C03659=1114.232,220.895,-68.578,-178.796,9.608,149.566
C03660=1114.228,221.144,-68.604,-178.794,9.611,149.566
C03661=1114.223,221.393,-68.631,-178.792,9.614,149.567
C03662=1114.219,221.641,-68.657,-178.789,9.617,149.567
C03663=1114.214,221.890,-68.684,-178.787,9.620,149.567
C03664=1114.210,222.138,-68.710,-178.784,9.623,149.567
C03665=1114.206,222.387,-68.737,-178.782,9.626,149.567
C03666=1114.202,222.635,-68.764,-178.779,9.629,149.567
C03667=1114.197,222.884,-68.790,-178.777,9.632,149.567
C03668=1114.193,223.132,-68.816,-178.774,9.635,149.567
C03669=1114.188,223.381,-68.843,-178.772,9.638,149.567
C03670=1114.184,223.629,-68.869,-178.769,9.642,149.567
C03671=1114.179,223.878,-68.896,-178.767,9.645,149.567
C03672=1114.175,224.126,-68.923,-178.764,9.648,149.567
C03673=1114.171,224.375,-68.950,-178.762,9.651,149.567
C03674=1114.166,224.623,-68.977,-178.759,9.654,149.567
C03675=1114.162,224.872,-69.003,-178.755,9.657,149.567
C03676=1114.157,225.120,-69.030,-178.753,9.661,149.567
C03677=1114.153,225.369,-69.057,-178.750,9.664,149.567
C03678=1114.150,225.582,-69.080,-178.749,9.666,149.567
C03679=1114.146,225.795,-69.102,-178.746,9.669,149.568
C03680=1114.142,226.008,-69.126,-178.744,9.671,149.568
C03681=1114.138,226.222,-69.149,-178.741,9.674,149.567
C03682=1114.135,226.435,-69.172,-178.739,9.677,149.568
C03683=1114.131,226.648,-69.194,-178.737,9.680,149.568
C03684=1114.127,226.861,-69.218,-178.735,9.682,149.568
C03685=1114.123,227.074,-69.241,-178.732,9.685,149.568
C03686=1114.119,227.323,-69.268,-178.729,9.688,149.568
C03687=1114.114,227.572,-69.294,-178.727,9.691,149.568
C03688=1114.110,227.820,-69.321,-178.724,9.694,149.568
C03689=1114.105,228.069,-69.348,-178.721,9.697,149.568
C03690=1114.101,228.317,-69.375,-178.718,9.700,149.567
C03691=1114.097,228.565,-69.403,-178.715,9.703,149.568
C03692=1114.093,228.814,-69.430,-178.712,9.706,149.567
C03693=1114.088,229.062,-69.457,-178.710,9.709,149.568
C03694=1114.084,229.311,-69.484,-178.707,9.712,149.567
C03695=1114.080,229.559,-69.511,-178.704,9.715,149.567
C03696=1114.075,229.808,-69.538,-178.701,9.719,149.567
C03697=1114.070,230.056,-69.565,-178.698,9.721,149.567
C03698=1114.066,230.305,-69.592,-178.695,9.724,149.567
C03699=1114.062,230.553,-69.619,-178.692,9.727,149.567
C03700=1114.058,230.802,-69.646,-178.689,9.730,149.567
C03701=1114.053,231.050,-69.673,-178.686,9.733,149.567
C03702=1114.049,231.298,-69.701,-178.684,9.736,149.567
C03703=1114.045,231.547,-69.728,-178.680,9.739,149.567
C03704=1114.040,231.796,-69.755,-178.677,9.742,149.567
C03705=1114.036,232.044,-69.781,-178.674,9.745,149.567
C03706=1114.032,232.292,-69.809,-178.672,9.748,149.566
C03707=1114.028,232.541,-69.837,-178.669,9.751,149.567
C03708=1114.023,232.790,-69.864,-178.666,9.754,149.566
C03709=1114.018,233.038,-69.891,-178.663,9.756,149.566
C03710=1114.014,233.286,-69.919,-178.661,9.758,149.566
C03711=1114.010,233.535,-69.946,-178.658,9.761,149.566
C03712=1114.005,233.784,-69.973,-178.655,9.764,149.566
C03713=1114.001,234.032,-70.001,-178.652,9.767,149.566
C03714=1113.997,234.281,-70.028,-178.649,9.770,149.566
C03715=1113.992,234.529,-70.055,-178.646,9.772,149.566
C03716=1113.989,234.777,-70.083,-178.644,9.775,149.566
C03717=1113.984,235.025,-70.110,-178.641,9.778,149.565
C03718=1113.980,235.274,-70.138,-178.639,9.780,149.566
C03719=1113.975,235.522,-70.165,-178.636,9.783,149.565
C03720=1113.971,235.771,-70.192,-178.633,9.786,149.565
C03721=1113.967,236.020,-70.220,-178.630,9.788,149.565
C03722=1113.962,236.268,-70.247,-178.627,9.791,149.565
C03723=1113.958,236.516,-70.275,-178.625,9.794,149.565
C03724=1113.954,236.765,-70.302,-178.622,9.796,149.565
C03725=1113.950,237.013,-70.330,-178.619,9.799,149.565
C03726=1113.944,237.262,-70.358,-178.617,9.801,149.565
C03727=1113.941,237.510,-70.386,-178.614,9.804,149.565
C03728=1113.936,237.759,-70.413,-178.611,9.807,149.565
C03729=1113.932,238.007,-70.441,-178.608,9.810,149.565
C03730=1113.927,238.256,-70.468,-178.606,9.812,149.564
C03731=1113.923,238.504,-70.496,-178.603,9.814,149.564
C03732=1113.919,238.752,-70.524,-178.601,9.816,149.564
C03733=1113.915,239.001,-70.551,-178.598,9.819,149.564
C03734=1113.911,239.214,-70.575,-178.596,9.821,149.564
C03735=1113.907,239.427,-70.598,-178.594,9.823,149.564
C03736=1113.903,239.640,-70.623,-178.592,9.826,149.564
C03737=1113.899,239.853,-70.646,-178.589,9.828,149.564
C03738=1113.896,240.066,-70.670,-178.587,9.831,149.564
C03739=1113.892,240.279,-70.694,-178.585,9.833,149.564
C03740=1113.889,240.492,-70.718,-178.583,9.835,149.564
C03741=1113.885,240.705,-70.742,-178.580,9.837,149.564
C03742=1113.880,240.954,-70.769,-178.578,9.839,149.564
C03743=1113.876,241.202,-70.797,-178.576,9.842,149.564
C03744=1113.872,241.450,-70.825,-178.573,9.844,149.564
C03745=1113.868,241.699,-70.853,-178.571,9.847,149.564
C03746=1113.863,241.947,-70.880,-178.568,9.849,149.563
C03747=1113.859,242.195,-70.908,-178.566,9.852,149.564
C03748=1113.855,242.444,-70.937,-178.564,9.854,149.563
C03749=1113.850,242.692,-70.965,-178.561,9.857,149.563
C03750=1113.846,242.941,-70.992,-178.559,9.859,149.563
C03751=1113.842,243.189,-71.020,-178.556,9.863,149.563
C03752=1113.837,243.438,-71.049,-178.554,9.864,149.563
C03753=1113.833,243.686,-71.076,-178.551,9.868,149.563
C03754=1113.829,243.934,-71.104,-178.549,9.870,149.563
C03755=1113.825,244.183,-71.131,-178.547,9.873,149.563
C03756=1113.820,244.432,-71.160,-178.545,9.875,149.563
C03757=1113.816,244.679,-71.188,-178.542,9.878,149.563
C03758=1113.812,244.928,-71.216,-178.540,9.880,149.563
C03759=1113.808,245.176,-71.244,-178.538,9.882,149.563
C03760=1113.803,245.425,-71.273,-178.535,9.886,149.563
C03761=1113.799,245.673,-71.300,-178.533,9.888,149.564
C03762=1113.795,245.921,-71.329,-178.531,9.891,149.563
C03763=1113.790,246.169,-71.357,-178.529,9.893,149.563
C03764=1113.786,246.418,-71.385,-178.526,9.896,149.564
C03765=1113.782,246.666,-71.413,-178.524,9.898,149.564
C03766=1113.777,246.915,-71.441,-178.522,9.901,149.564
C03767=1113.773,247.163,-71.469,-178.520,9.904,149.564
C03768=1113.769,247.412,-71.497,-178.518,9.906,149.564
C03769=1113.764,247.660,-71.525,-178.514,9.910,149.564
C03770=1113.760,247.909,-71.553,-178.511,9.913,149.564
C03771=1113.755,248.156,-71.582,-178.507,9.918,149.564
C03772=1113.752,248.405,-71.611,-178.503,9.921,149.563
C03773=1113.748,248.653,-71.639,-178.499,9.924,149.563
C03774=1113.743,248.902,-71.667,-178.495,9.927,149.563
C03775=1113.739,249.150,-71.695,-178.491,9.931,149.563
C03776=1113.734,249.398,-71.724,-178.487,9.934,149.562
C03777=1113.730,249.647,-71.752,-178.484,9.937,149.562
C03778=1113.726,249.896,-71.780,-178.481,9.940,149.562
C03779=1113.721,250.144,-71.808,-178.477,9.942,149.562
C03780=1113.717,250.392,-71.838,-178.474,9.946,149.562
C03781=1113.713,250.640,-71.865,-178.470,9.948,149.561
C03782=1113.708,250.889,-71.894,-178.467,9.951,149.561
C03783=1113.705,251.137,-71.922,-178.464,9.954,149.561
C03784=1113.700,251.385,-71.951,-178.461,9.956,149.561
C03785=1113.696,251.633,-71.980,-178.458,9.959,149.561
C03786=1113.692,251.882,-72.008,-178.455,9.961,149.560
C03787=1113.687,252.130,-72.036,-178.452,9.964,149.560
C03788=1113.683,252.378,-72.066,-178.449,9.967,149.560
C03789=1113.679,252.627,-72.094,-178.446,9.969,149.560
C03790=1113.675,252.840,-72.119,-178.444,9.971,149.560
C03791=1113.672,253.052,-72.143,-178.442,9.973,149.560
C03792=1113.668,253.266,-72.168,-178.440,9.975,149.560
C03793=1113.664,253.479,-72.192,-178.437,9.977,149.560
C03794=1113.660,253.691,-72.216,-178.435,9.979,149.559
C03795=1113.657,253.905,-72.241,-178.433,9.981,149.559
C03796=1113.653,254.117,-72.266,-178.431,9.982,149.559
C03797=1113.649,254.330,-72.290,-178.429,9.984,149.559
C03798=1113.645,254.578,-72.319,-178.427,9.987,149.559
C03799=1113.641,254.827,-72.348,-178.425,9.989,149.559
C03800=1113.637,255.076,-72.377,-178.423,9.991,149.559
C03801=1113.633,255.323,-72.405,-178.421,9.993,149.559
C03802=1113.628,255.572,-72.434,-178.420,9.995,149.559
C03803=1113.624,255.821,-72.463,-178.418,9.997,149.559
C03804=1113.620,256.068,-72.491,-178.416,10.000,149.559
C03805=1113.615,256.317,-72.520,-178.413,10.002,149.559
C03806=1113.611,256.565,-72.549,-178.410,10.005,149.559
C03807=1113.607,256.814,-72.578,-178.408,10.007,149.559
C03808=1113.602,257.061,-72.607,-178.405,10.010,149.559
C03809=1113.598,257.310,-72.635,-178.402,10.013,149.559
C03810=1113.594,257.558,-72.665,-178.399,10.016,149.559
C03811=1113.590,257.806,-72.694,-178.396,10.018,149.559
C03812=1113.585,258.054,-72.722,-178.394,10.022,149.559
C03813=1113.581,258.303,-72.752,-178.391,10.024,149.559
C03814=1113.577,258.551,-72.780,-178.388,10.027,149.559
C03815=1113.573,258.800,-72.809,-178.385,10.030,149.559
C03816=1113.569,259.048,-72.839,-178.382,10.033,149.558
C03817=1113.564,259.296,-72.867,-178.379,10.035,149.558
C03818=1113.560,259.544,-72.896,-178.376,10.038,149.558
C03819=1113.556,259.793,-72.925,-178.374,10.041,149.558
C03820=1113.552,260.041,-72.954,-178.371,10.044,149.558
C03821=1113.548,260.289,-72.983,-178.368,10.047,149.558
C03822=1113.543,260.537,-73.013,-178.365,10.049,149.558
C03823=1113.538,260.786,-73.041,-178.362,10.052,149.558
C03824=1113.535,261.034,-73.070,-178.359,10.055,149.558
C03825=1113.531,261.282,-73.100,-178.356,10.058,149.558
C03826=1113.526,261.530,-73.129,-178.353,10.060,149.558
C03827=1113.522,261.779,-73.158,-178.350,10.063,149.558
C03828=1113.518,262.027,-73.187,-178.347,10.066,149.557
C03829=1113.513,262.275,-73.216,-178.344,10.068,149.557
C03830=1113.509,262.523,-73.246,-178.341,10.071,149.557
C03831=1113.505,262.772,-73.275,-178.338,10.074,149.557
C03832=1113.501,263.020,-73.303,-178.335,10.077,149.557
C03833=1113.497,263.268,-73.333,-178.332,10.080,149.557
C03834=1113.493,263.517,-73.362,-178.328,10.083,149.556
C03835=1113.488,263.765,-73.392,-178.325,10.085,149.556
C03836=1113.484,264.013,-73.421,-178.322,10.088,149.556
C03837=1113.479,264.261,-73.450,-178.319,10.091,149.556
C03838=1113.475,264.509,-73.480,-178.316,10.093,149.556
C03839=1113.471,264.757,-73.509,-178.313,10.096,149.556
C03840=1113.467,265.006,-73.539,-178.311,10.098,149.556
C03841=1113.463,265.254,-73.568,-178.308,10.101,149.555
C03842=1113.458,265.502,-73.598,-178.305,10.104,149.555
C03843=1113.454,265.750,-73.627,-178.303,10.106,149.555
C03844=1113.450,265.999,-73.656,-178.300,10.108,149.555
C03845=1113.446,266.247,-73.686,-178.297,10.111,149.555
C03846=1113.442,266.460,-73.711,-178.294,10.113,149.555
C03847=1113.438,266.672,-73.737,-178.292,10.115,149.555
C03848=1113.434,266.885,-73.761,-178.290,10.117,149.555
C03849=1113.431,267.098,-73.787,-178.288,10.119,149.555
C03850=1113.427,267.311,-73.813,-178.285,10.122,149.554
C03851=1113.424,267.523,-73.838,-178.282,10.124,149.554
C03852=1113.420,267.737,-73.863,-178.280,10.126,149.554
C03853=1113.416,267.949,-73.889,-178.278,10.128,149.554
C03854=1113.412,268.197,-73.918,-178.275,10.131,149.554
C03855=1113.408,268.445,-73.948,-178.272,10.134,149.554
C03856=1113.404,268.694,-73.977,-178.270,10.136,149.554
C03857=1113.399,268.942,-74.007,-178.267,10.138,149.554
C03858=1113.395,269.190,-74.036,-178.264,10.141,149.554
C03859=1113.391,269.438,-74.066,-178.261,10.144,149.554
C03860=1113.387,269.686,-74.096,-178.259,10.146,149.553
C03861=1113.382,269.935,-74.126,-178.256,10.149,149.553
C03862=1113.378,270.183,-74.155,-178.253,10.151,149.553
C03863=1113.374,270.431,-74.185,-178.250,10.154,149.553
C03864=1113.370,270.679,-74.215,-178.247,10.156,149.553
C03865=1113.366,270.927,-74.244,-178.244,10.158,149.553
C03866=1113.362,271.176,-74.275,-178.241,10.161,149.553
C03867=1113.358,271.424,-74.305,-178.238,10.164,149.553
C03868=1113.354,271.672,-74.334,-178.235,10.167,149.552
C03869=1113.349,271.921,-74.364,-178.233,10.170,149.552
C03870=1113.345,272.168,-74.394,-178.230,10.172,149.552
C03871=1113.341,272.417,-74.424,-178.227,10.174,149.552
C03872=1113.336,272.665,-74.453,-178.224,10.177,149.552
C03873=1113.333,272.913,-74.484,-178.221,10.180,149.552
C03874=1113.328,273.161,-74.513,-178.219,10.183,149.552
C03875=1113.323,273.410,-74.543,-178.216,10.185,149.552
C03876=1113.320,273.657,-74.573,-178.213,10.188,149.552
C03877=1113.315,273.906,-74.603,-178.210,10.191,149.552
C03878=1113.312,274.154,-74.633,-178.206,10.193,149.551
C03879=1113.307,274.402,-74.663,-178.204,10.195,149.551
C03880=1113.303,274.650,-74.693,-178.201,10.198,149.551
C03881=1113.299,274.898,-74.723,-178.198,10.201,149.551
C03882=1113.294,275.146,-74.754,-178.195,10.204,149.551
C03883=1113.290,275.395,-74.783,-178.192,10.206,149.551
C03884=1113.286,275.642,-74.813,-178.189,10.209,149.551
C03885=1113.282,275.892,-74.844,-178.186,10.211,149.550
C03886=1113.278,276.139,-74.874,-178.183,10.214,149.550
C03887=1113.274,276.387,-74.903,-178.180,10.217,149.550
C03888=1113.269,276.635,-74.934,-178.177,10.220,149.550
C03889=1113.266,276.883,-74.964,-178.174,10.223,149.550
C03890=1113.261,277.131,-74.994,-178.171,10.225,149.550
C03891=1113.257,277.380,-75.025,-178.168,10.228,149.550
C03892=1113.253,277.628,-75.055,-178.165,10.230,149.550
C03893=1113.249,277.876,-75.085,-178.163,10.232,149.549
C03894=1113.245,278.124,-75.115,-178.159,10.235,149.549
C03895=1113.240,278.372,-75.146,-178.156,10.238,149.549
C03896=1113.237,278.621,-75.176,-178.154,10.240,149.549
C03897=1113.233,278.868,-75.206,-178.150,10.243,149.549
C03898=1113.228,279.116,-75.237,-178.147,10.246,149.549
C03899=1113.224,279.365,-75.266,-178.144,10.248,149.548
C03900=1113.220,279.613,-75.297,-178.141,10.251,149.548
C03901=1113.216,279.861,-75.327,-178.138,10.253,149.548
C03902=1113.212,280.074,-75.354,-178.135,10.256,149.548
C03903=1113.208,280.286,-75.380,-178.133,10.258,149.548
C03904=1113.205,280.499,-75.405,-178.130,10.260,149.548
C03905=1113.201,280.712,-75.432,-178.127,10.263,149.547
C03906=1113.198,280.924,-75.459,-178.125,10.265,149.547
C03907=1113.194,281.136,-75.484,-178.122,10.267,149.547
C03908=1113.190,281.349,-75.511,-178.120,10.269,149.547
C03909=1113.187,281.562,-75.536,-178.116,10.272,149.547
C03910=1113.183,281.810,-75.567,-178.114,10.274,149.547
C03911=1113.179,282.059,-75.598,-178.111,10.276,149.546
C03912=1113.174,282.306,-75.628,-178.108,10.279,149.546
C03913=1113.170,282.554,-75.659,-178.105,10.282,149.546
C03914=1113.166,282.802,-75.689,-178.101,10.284,149.546
C03915=1113.162,283.051,-75.721,-178.098,10.287,149.546
C03916=1113.158,283.299,-75.750,-178.095,10.289,149.546
C03917=1113.153,283.547,-75.781,-178.092,10.292,149.546
C03918=1113.150,283.795,-75.811,-178.090,10.294,149.545
C03919=1113.145,284.043,-75.842,-178.087,10.296,149.545
C03920=1113.140,284.291,-75.873,-178.084,10.299,149.545
C03921=1113.137,284.540,-75.903,-178.080,10.302,149.545
C03922=1113.133,284.787,-75.935,-178.077,10.304,149.545
C03923=1113.128,285.035,-75.966,-178.074,10.307,149.544
C03924=1113.125,285.283,-75.996,-178.071,10.310,149.544
C03925=1113.120,285.531,-76.027,-178.068,10.312,149.544
C03926=1113.116,285.779,-76.058,-178.065,10.315,149.544
C03927=1113.112,286.028,-76.089,-178.062,10.317,149.544
C03928=1113.108,286.275,-76.119,-178.059,10.319,149.544
C03929=1113.104,286.524,-76.150,-178.056,10.322,149.543
C03930=1113.099,286.772,-76.181,-178.053,10.324,149.543
C03931=1113.096,287.019,-76.212,-178.050,10.327,149.543
C03932=1113.092,287.268,-76.243,-178.047,10.330,149.543
C03933=1113.087,287.516,-76.274,-178.044,10.332,149.543
C03934=1113.083,287.764,-76.305,-178.041,10.335,149.543
C03935=1113.078,288.012,-76.336,-178.038,10.337,149.542
C03936=1113.075,288.259,-76.366,-178.035,10.340,149.542
C03937=1113.071,288.508,-76.398,-178.032,10.342,149.542
C03938=1113.066,288.756,-76.428,-178.029,10.345,149.542
C03939=1113.062,289.005,-76.459,-178.026,10.347,149.542
C03940=1113.058,289.252,-76.491,-178.023,10.350,149.542
C03941=1113.055,289.500,-76.521,-178.020,10.353,149.541
C03942=1113.050,289.748,-76.552,-178.016,10.355,149.541
C03943=1113.046,289.996,-76.584,-178.013,10.358,149.541
C03944=1113.042,290.244,-76.615,-178.011,10.359,149.541
C03945=1113.037,290.492,-76.646,-178.008,10.362,149.541
C03946=1113.033,290.740,-76.677,-178.004,10.365,149.540
C03947=1113.029,290.988,-76.708,-178.001,10.367,149.540
C03948=1113.026,291.236,-76.739,-177.998,10.370,149.540
C03949=1113.021,291.484,-76.770,-177.995,10.373,149.540
C03950=1113.017,291.733,-76.801,-177.992,10.375,149.540
C03951=1113.013,291.980,-76.833,-177.989,10.378,149.540
C03952=1113.009,292.229,-76.864,-177.986,10.381,149.540
C03953=1113.005,292.476,-76.895,-177.983,10.382,149.539
C03954=1113.001,292.725,-76.927,-177.980,10.385,149.539
C03955=1112.997,292.973,-76.958,-177.977,10.387,149.539
C03956=1112.992,293.221,-76.989,-177.974,10.390,149.539
C03957=1112.989,293.469,-77.021,-177.971,10.393,149.539
C03958=1112.985,293.681,-77.048,-177.968,10.395,149.538
C03959=1112.982,293.894,-77.074,-177.965,10.397,149.538
C03960=1112.978,294.106,-77.101,-177.963,10.399,149.538
C03961=1112.974,294.319,-77.129,-177.960,10.401,149.538
C03962=1112.971,294.531,-77.155,-177.958,10.404,149.538
C03963=1112.968,294.743,-77.182,-177.955,10.406,149.538
C03964=1112.964,294.956,-77.210,-177.953,10.408,149.538
C03965=1112.961,295.169,-77.235,-177.950,10.410,149.537
C03966=1112.956,295.416,-77.267,-177.947,10.413,149.537
C03967=1112.953,295.664,-77.299,-177.944,10.415,149.537
C03968=1112.947,295.912,-77.330,-177.941,10.417,149.537
C03969=1112.944,296.160,-77.362,-177.938,10.420,149.537
C03970=1112.940,296.408,-77.394,-177.935,10.423,149.537
C03971=1112.935,296.656,-77.425,-177.932,10.425,149.536
C03972=1112.932,296.904,-77.456,-177.928,10.428,149.536
C03973=1112.927,297.152,-77.488,-177.926,10.431,149.536
C03974=1112.924,297.400,-77.520,-177.922,10.433,149.536
C03975=1112.920,297.648,-77.551,-177.919,10.436,149.536
C03976=1112.915,297.896,-77.582,-177.917,10.437,149.535
C03977=1112.911,298.144,-77.615,-177.914,10.440,149.535
C03978=1112.907,298.392,-77.647,-177.910,10.443,149.535
C03979=1112.903,298.640,-77.678,-177.907,10.445,149.535
C03980=1112.899,298.888,-77.709,-177.904,10.448,149.535
C03981=1112.895,299.136,-77.741,-177.901,10.451,149.535
C03982=1112.891,299.384,-77.773,-177.898,10.453,149.534
C03983=1112.886,299.632,-77.805,-177.895,10.456,149.534
C03984=1112.883,299.880,-77.837,-177.892,10.458,149.534
C03985=1112.878,300.127,-77.868,-177.889,10.461,149.534
C03986=1112.875,300.375,-77.900,-177.886,10.463,149.534
C03987=1112.871,300.623,-77.932,-177.883,10.465,149.534
C03988=1112.866,300.871,-77.964,-177.880,10.468,149.533
C03989=1112.862,301.119,-77.996,-177.877,10.471,149.533
C03990=1112.858,301.367,-78.028,-177.873,10.473,149.533
C03991=1112.853,301.615,-78.060,-177.870,10.476,149.533
C03992=1112.850,301.863,-78.092,-177.867,10.478,149.533
C03993=1112.846,302.111,-78.124,-177.864,10.481,149.533
C03994=1112.842,302.358,-78.155,-177.861,10.483,149.532
C03995=1112.837,302.607,-78.188,-177.859,10.485,149.532
C03996=1112.833,302.855,-78.219,-177.855,10.488,149.532
C03997=1112.830,303.103,-78.251,-177.852,10.491,149.532
C03998=1112.825,303.350,-78.283,-177.849,10.493,149.532
C03999=1112.821,303.598,-78.315,-177.846,10.496,149.532
C04000=1112.817,303.847,-78.348,-177.843,10.498,149.531
C04001=1112.813,304.095,-78.379,-177.840,10.501,149.531
C04002=1112.809,304.342,-78.411,-177.836,10.503,149.531
C04003=1112.804,304.590,-78.443,-177.833,10.506,149.531
C04004=1112.801,304.838,-78.476,-177.830,10.509,149.531
C04005=1112.797,305.086,-78.508,-177.827,10.510,149.530
C04006=1112.792,305.333,-78.540,-177.825,10.513,149.530
C04007=1112.788,305.582,-78.572,-177.821,10.516,149.530
C04008=1112.784,305.830,-78.604,-177.818,10.518,149.530
C04009=1112.780,306.077,-78.637,-177.815,10.521,149.530
C04010=1112.776,306.326,-78.669,-177.812,10.523,149.530
C04011=1112.772,306.573,-78.701,-177.809,10.526,149.529
C04012=1112.768,306.821,-78.732,-177.806,10.529,149.529
C04013=1112.764,307.069,-78.766,-177.802,10.531,149.529
C04014=1112.760,307.281,-78.793,-177.800,10.533,149.529
C04015=1112.757,307.493,-78.821,-177.798,10.535,149.529
C04016=1112.754,307.706,-78.848,-177.794,10.538,149.528
C04017=1112.750,307.918,-78.876,-177.792,10.540,149.528
C04018=1112.747,308.131,-78.903,-177.790,10.542,149.528
C04019=1112.742,308.343,-78.932,-177.787,10.544,149.528
C04020=1112.739,308.556,-78.959,-177.784,10.546,149.528
C04021=1112.736,308.768,-78.987,-177.782,10.548,149.528
C04022=1112.732,309.016,-79.019,-177.779,10.550,149.528
C04023=1112.728,309.264,-79.052,-177.776,10.553,149.527
C04024=1112.724,309.511,-79.084,-177.772,10.556,149.527
C04025=1112.719,309.759,-79.116,-177.769,10.558,149.527
C04026=1112.716,310.007,-79.149,-177.766,10.561,149.527
C04027=1112.712,310.255,-79.181,-177.763,10.563,149.527
C04028=1112.707,310.503,-79.214,-177.760,10.566,149.527
C04029=1112.704,310.751,-79.246,-177.757,10.568,149.526
C04030=1112.700,310.999,-79.279,-177.754,10.570,149.526
C04031=1112.696,311.247,-79.311,-177.751,10.573,149.526
C04032=1112.692,311.494,-79.345,-177.748,10.576,149.526
C04033=1112.687,311.743,-79.377,-177.745,10.578,149.526
C04034=1112.684,311.990,-79.410,-177.741,10.581,149.525
C04035=1112.679,312.237,-79.442,-177.738,10.583,149.525
C04036=1112.675,312.485,-79.475,-177.735,10.586,149.525
C04037=1112.671,312.733,-79.507,-177.732,10.589,149.525
C04038=1112.667,312.981,-79.540,-177.729,10.591,149.525
C04039=1112.663,313.229,-79.573,-177.726,10.594,149.525
C04040=1112.659,313.476,-79.605,-177.723,10.595,149.524
C04041=1112.655,313.725,-79.638,-177.720,10.598,149.524
C04042=1112.651,313.972,-79.671,-177.717,10.601,149.524
C04043=1112.647,314.220,-79.704,-177.714,10.603,149.524
C04044=1112.643,314.468,-79.737,-177.711,10.606,149.524
C04045=1112.639,314.716,-79.769,-177.707,10.608,149.523
C04046=1112.635,314.963,-79.802,-177.704,10.611,149.523
C04047=1112.631,315.211,-79.835,-177.701,10.613,149.523
C04048=1112.627,315.459,-79.868,-177.698,10.616,149.523
C04049=1112.623,315.707,-79.901,-177.695,10.619,149.523
C04050=1112.619,315.955,-79.933,-177.692,10.620,149.523
C04051=1112.615,316.202,-79.966,-177.689,10.623,149.522
C04052=1112.611,316.450,-79.999,-177.686,10.626,149.522
C04053=1112.607,316.698,-80.033,-177.683,10.628,149.522
C04054=1112.603,316.946,-80.066,-177.680,10.631,149.522
C04055=1112.599,317.194,-80.098,-177.676,10.633,149.522
C04056=1112.595,317.441,-80.131,-177.673,10.636,149.522
C04057=1112.591,317.690,-80.164,-177.670,10.638,149.521
C04058=1112.587,317.937,-80.197,-177.667,10.641,149.521
C04059=1112.583,318.185,-80.231,-177.664,10.644,149.521
C04060=1112.579,318.433,-80.264,-177.660,10.646,149.521
C04061=1112.575,318.680,-80.296,-177.658,10.648,149.521
C04062=1112.571,318.928,-80.329,-177.655,10.651,149.520
C04063=1112.567,319.176,-80.363,-177.652,10.653,149.520
C04064=1112.563,319.424,-80.396,-177.649,10.656,149.520
C04065=1112.559,319.671,-80.429,-177.645,10.658,149.520
C04066=1112.555,319.919,-80.462,-177.642,10.661,149.520
C04067=1112.551,320.167,-80.496,-177.639,10.663,149.520
C04068=1112.547,320.415,-80.529,-177.636,10.666,149.519
C04069=1112.544,320.663,-80.561,-177.633,10.669,149.519
C04070=1112.540,320.875,-80.590,-177.630,10.670,149.519
C04071=1112.537,321.087,-80.618,-177.628,10.672,149.519
C04072=1112.533,321.299,-80.647,-177.624,10.675,149.519
C04073=1112.530,321.511,-80.676,-177.622,10.677,149.518
C04074=1112.526,321.724,-80.704,-177.620,10.679,149.518
C04075=1112.523,321.936,-80.732,-177.617,10.681,149.518
C04076=1112.519,322.148,-80.761,-177.614,10.683,149.518
C04077=1112.516,322.360,-80.790,-177.612,10.685,149.518
C04078=1112.513,322.608,-80.823,-177.609,10.688,149.518
C04079=1112.508,322.856,-80.856,-177.605,10.690,149.517
C04080=1112.504,323.103,-80.889,-177.602,10.693,149.517
C04081=1112.500,323.351,-80.923,-177.599,10.695,149.517
C04082=1112.496,323.598,-80.956,-177.596,10.698,149.517
C04083=1112.493,323.847,-80.990,-177.593,10.701,149.517
C04084=1112.489,324.094,-81.023,-177.590,10.703,149.517
C04085=1112.485,324.342,-81.056,-177.586,10.705,149.516
C04086=1112.480,324.590,-81.091,-177.583,10.708,149.516
C04087=1112.476,324.837,-81.124,-177.581,10.710,149.516
C04088=1112.472,325.086,-81.157,-177.577,10.712,149.516
C04089=1112.468,325.333,-81.191,-177.574,10.715,149.516
C04090=1112.464,325.581,-81.224,-177.571,10.718,149.515
C04091=1112.460,325.828,-81.258,-177.568,10.720,149.515
C04092=1112.457,326.076,-81.292,-177.565,10.723,149.515
C04093=1112.453,326.324,-81.325,-177.561,10.725,149.515
C04094=1112.449,326.571,-81.359,-177.558,10.728,149.515
C04095=1112.444,326.819,-81.393,-177.555,10.730,149.515
C04096=1112.441,327.067,-81.426,-177.552,10.733,149.514
C04097=1112.437,327.315,-81.460,-177.549,10.735,149.514
C04098=1112.433,327.562,-81.493,-177.546,10.737,149.514
C04099=1112.429,327.809,-81.527,-177.543,10.740,149.514
C04100=1112.425,328.058,-81.561,-177.540,10.742,149.514
C04101=1112.421,328.305,-81.595,-177.537,10.745,149.513
C04102=1112.417,328.553,-81.628,-177.533,10.747,149.513
C04103=1112.413,328.800,-81.662,-177.530,10.750,149.513
C04104=1112.409,329.048,-81.696,-177.527,10.753,149.513
C04105=1112.405,329.296,-81.730,-177.524,10.755,149.513
C04106=1112.401,329.543,-81.764,-177.521,10.758,149.512
C04107=1112.397,329.791,-81.797,-177.518,10.760,149.512
C04108=1112.393,330.039,-81.831,-177.515,10.762,149.512
C04109=1112.389,330.287,-81.865,-177.512,10.765,149.512
C04110=1112.385,330.534,-81.899,-177.509,10.767,149.512
C04111=1112.381,330.781,-81.933,-177.505,10.770,149.512
C04112=1112.377,331.030,-81.967,-177.502,10.772,149.511
C04113=1112.373,331.277,-82.001,-177.499,10.775,149.511
C04114=1112.370,331.524,-82.035,-177.496,10.777,149.511
C04115=1112.365,331.772,-82.069,-177.492,10.780,149.511
C04116=1112.361,332.020,-82.103,-177.489,10.782,149.511
C04117=1112.358,332.267,-82.137,-177.486,10.785,149.511
C04118=1112.354,332.516,-82.172,-177.484,10.787,149.510
C04119=1112.349,332.763,-82.205,-177.480,10.789,149.510
C04120=1112.346,333.010,-82.239,-177.477,10.792,149.510
C04121=1112.342,333.258,-82.274,-177.474,10.794,149.510
C04122=1112.338,333.506,-82.307,-177.471,10.797,149.509
C04123=1112.334,333.753,-82.341,-177.467,10.799,149.509
C04124=1112.330,334.001,-82.375,-177.464,10.802,149.509
C04125=1112.326,334.249,-82.409,-177.461,10.805,149.509
C04126=1112.323,334.461,-82.439,-177.458,10.806,149.509
C04127=1112.319,334.673,-82.468,-177.456,10.808,149.509
C04128=1112.316,334.885,-82.498,-177.453,10.811,149.508
C04129=1112.312,335.097,-82.527,-177.451,10.813,149.508
C04130=1112.309,335.310,-82.556,-177.448,10.816,149.508
C04131=1112.306,335.521,-82.585,-177.445,10.817,149.508
C04132=1112.303,335.733,-82.614,-177.443,10.819,149.508
C04133=1112.299,335.945,-82.644,-177.439,10.822,149.508
C04134=1112.295,336.193,-82.679,-177.437,10.823,149.507
C04135=1112.292,336.441,-82.713,-177.434,10.826,149.507
C04136=1112.287,336.688,-82.747,-177.430,10.829,149.507
C04137=1112.284,336.936,-82.781,-177.427,10.831,149.507
C04138=1112.279,337.183,-82.816,-177.424,10.833,149.507
C04139=1112.276,337.431,-82.850,-177.421,10.836,149.507
C04140=1112.271,337.679,-82.885,-177.418,10.839,149.506
C04141=1112.268,337.926,-82.919,-177.414,10.841,149.506
C04142=1112.264,338.174,-82.953,-177.411,10.844,149.506
C04143=1112.260,338.422,-82.988,-177.408,10.846,149.506
C04144=1112.256,338.669,-83.022,-177.405,10.849,149.506
C04145=1112.251,338.916,-83.056,-177.402,10.851,149.505
C04146=1112.248,339.164,-83.091,-177.399,10.853,149.505
C04147=1112.244,339.411,-83.126,-177.396,10.856,149.505
C04148=1112.240,339.659,-83.161,-177.392,10.858,149.505
C04149=1112.237,339.907,-83.195,-177.389,10.861,149.505
C04150=1112.232,340.154,-83.229,-177.386,10.863,149.504
C04151=1112.229,340.402,-83.264,-177.382,10.866,149.504
C04152=1112.225,340.649,-83.299,-177.380,10.868,149.504
C04153=1112.221,340.897,-83.334,-177.376,10.871,149.504
C04154=1112.216,341.145,-83.368,-177.373,10.873,149.504
C04155=1112.213,341.392,-83.402,-177.370,10.875,149.503
C04156=1112.208,341.639,-83.438,-177.367,10.878,149.503
C04157=1112.205,341.887,-83.472,-177.364,10.880,149.503
C04158=1112.201,342.134,-83.506,-177.361,10.883,149.503
C04159=1112.197,342.382,-83.542,-177.357,10.885,149.503
C04160=1112.193,342.630,-83.577,-177.354,10.888,149.502
C04161=1112.189,342.877,-83.611,-177.351,10.890,149.502
C04162=1112.186,343.125,-83.646,-177.348,10.893,149.502
C04163=1112.181,343.372,-83.681,-177.345,10.895,149.502
C04164=1112.177,343.620,-83.715,-177.341,10.898,149.502
C04165=1112.173,343.868,-83.751,-177.338,10.900,149.501
C04166=1112.170,344.115,-83.785,-177.336,10.902,149.501
C04167=1112.166,344.362,-83.820,-177.332,10.905,149.501
C04168=1112.161,344.610,-83.855,-177.329,10.907,149.501
C04169=1112.157,344.858,-83.890,-177.326,10.910,149.501
C04170=1112.154,345.105,-83.925,-177.322,10.912,149.500
C04171=1112.150,345.352,-83.959,-177.319,10.915,149.500
C04172=1112.146,345.600,-83.995,-177.316,10.917,149.500
C04173=1112.142,345.848,-84.029,-177.313,10.920,149.500
C04174=1112.138,346.095,-84.065,-177.310,10.922,149.500
C04175=1112.134,346.343,-84.099,-177.306,10.925,149.499
C04176=1112.131,346.590,-84.134,-177.304,10.927,149.499
C04177=1112.127,346.837,-84.170,-177.301,10.929,149.499
C04178=1112.123,347.085,-84.204,-177.297,10.932,149.499
C04179=1112.119,347.333,-84.240,-177.294,10.934,149.499
C04180=1112.115,347.580,-84.274,-177.291,10.937,149.498
C04181=1112.111,347.828,-84.310,-177.287,10.939,149.498
C04182=1112.108,348.040,-84.340,-177.285,10.941,149.498
C04183=1112.105,348.251,-84.370,-177.282,10.943,149.498
C04184=1112.101,348.463,-84.401,-177.279,10.946,149.498
C04185=1112.098,348.676,-84.430,-177.277,10.947,149.498
C04186=1112.095,348.887,-84.461,-177.274,10.950,149.497
C04187=1112.091,349.100,-84.491,-177.271,10.952,149.497
C04188=1112.088,349.311,-84.521,-177.269,10.953,149.497
C04189=1112.084,349.523,-84.550,-177.266,10.956,149.497
C04190=1112.081,349.770,-84.586,-177.262,10.959,149.497
C04191=1112.077,350.018,-84.622,-177.259,10.961,149.496
C04192=1112.073,350.265,-84.657,-177.256,10.964,149.496
C04193=1112.069,350.513,-84.692,-177.252,10.966,149.496
C04194=1112.065,350.760,-84.727,-177.249,10.968,149.496
C04195=1112.061,351.008,-84.763,-177.246,10.971,149.496
C04196=1112.058,351.255,-84.798,-177.242,10.973,149.495
C04197=1112.054,351.502,-84.833,-177.239,10.976,149.495
C04198=1112.050,351.750,-84.869,-177.236,10.978,149.495
C04199=1112.046,351.998,-84.904,-177.233,10.981,149.495
C04200=1112.042,352.245,-84.939,-177.229,10.983,149.494
C04201=1112.039,352.493,-84.975,-177.226,10.986,149.494
C04202=1112.035,352.740,-85.010,-177.223,10.988,149.494
C04203=1112.031,352.987,-85.046,-177.219,10.991,149.494
C04204=1112.026,353.235,-85.082,-177.216,10.993,149.493
C04205=1112.023,353.482,-85.117,-177.212,10.995,149.493
C04206=1112.019,353.730,-85.153,-177.209,10.998,149.493
C04207=1112.015,353.977,-85.188,-177.206,11.000,149.493
C04208=1112.012,354.225,-85.224,-177.202,11.003,149.492
C04209=1112.007,354.472,-85.259,-177.199,11.005,149.492
C04210=1112.004,354.719,-85.295,-177.196,11.008,149.492
C04211=1112.000,354.967,-85.330,-177.192,11.010,149.492
C04212=1111.996,355.215,-85.366,-177.189,11.012,149.492
C04213=1111.992,355.462,-85.402,-177.185,11.015,149.491
C04214=1111.988,355.710,-85.437,-177.182,11.017,149.491
C04215=1111.985,355.957,-85.473,-177.179,11.020,149.491
C04216=1111.981,356.204,-85.509,-177.175,11.022,149.491
C04217=1111.977,356.451,-85.544,-177.172,11.024,149.490
C04218=1111.973,356.699,-85.581,-177.169,11.027,149.490
C04219=1111.969,356.946,-85.616,-177.166,11.029,149.490
C04220=1111.965,357.194,-85.652,-177.162,11.032,149.489
C04221=1111.962,357.441,-85.687,-177.159,11.034,149.489
C04222=1111.958,357.688,-85.723,-177.155,11.036,149.489
C04223=1111.954,357.936,-85.760,-177.152,11.039,149.489
C04224=1111.950,358.183,-85.795,-177.149,11.041,149.489
C04225=1111.947,358.431,-85.831,-177.145,11.044,149.488
C04226=1111.942,358.678,-85.868,-177.142,11.046,149.488
C04227=1111.939,358.925,-85.903,-177.138,11.048,149.488
C04228=1111.935,359.173,-85.939,-177.135,11.051,149.488
C04229=1111.932,359.420,-85.975,-177.132,11.053,149.487
C04230=1111.927,359.668,-86.011,-177.128,11.056,149.487
C04231=1111.924,359.915,-86.047,-177.125,11.058,149.487
C04232=1111.920,360.162,-86.083,-177.121,11.060,149.486
C04233=1111.916,360.410,-86.119,-177.118,11.063,149.486
C04234=1111.913,360.657,-86.155,-177.115,11.065,149.486
C04235=1111.909,360.904,-86.191,-177.111,11.068,149.486
C04236=1111.905,361.152,-86.227,-177.108,11.070,149.485
C04237=1111.901,361.399,-86.263,-177.104,11.073,149.485
C04238=1111.898,361.611,-86.294,-177.102,11.074,149.485
C04239=1111.895,361.822,-86.324,-177.098,11.077,149.485
C04240=1111.891,362.034,-86.356,-177.096,11.078,149.484
C04241=1111.888,362.246,-86.387,-177.093,11.080,149.484
C04242=1111.885,362.458,-86.418,-177.090,11.083,149.484
C04243=1111.882,362.670,-86.449,-177.088,11.085,149.484
C04244=1111.878,362.881,-86.480,-177.084,11.087,149.484
C04245=1111.875,363.093,-86.511,-177.082,11.089,149.483
C04246=1111.871,363.340,-86.547,-177.078,11.091,149.483
C04247=1111.868,363.588,-86.583,-177.075,11.093,149.483
C04248=1111.864,363.835,-86.620,-177.071,11.096,149.483
C04249=1111.860,364.082,-86.655,-177.068,11.098,149.482
C04250=1111.856,364.329,-86.692,-177.065,11.101,149.482
C04251=1111.853,364.577,-86.729,-177.061,11.103,149.482
C04252=1111.849,364.825,-86.765,-177.058,11.105,149.482
C04253=1111.845,365.072,-86.801,-177.054,11.108,149.481
C04254=1111.841,365.319,-86.838,-177.051,11.110,149.481
C04255=1111.838,365.566,-86.874,-177.048,11.113,149.481
C04256=1111.833,365.814,-86.911,-177.044,11.115,149.481
C04257=1111.830,366.060,-86.947,-177.041,11.117,149.480
C04258=1111.826,366.308,-86.983,-177.037,11.120,149.480
C04259=1111.822,366.555,-87.019,-177.034,11.122,149.480
C04260=1111.818,366.802,-87.056,-177.031,11.125,149.480
C04261=1111.815,367.050,-87.093,-177.028,11.127,149.480
C04262=1111.811,367.298,-87.129,-177.024,11.129,149.479
C04263=1111.807,367.545,-87.166,-177.021,11.132,149.479
C04264=1111.804,367.792,-87.202,-177.017,11.134,149.479
C04265=1111.800,368.039,-87.239,-177.014,11.137,149.479
C04266=1111.795,368.286,-87.276,-177.011,11.139,149.478
C04267=1111.793,368.534,-87.312,-177.007,11.142,149.478
C04268=1111.789,368.781,-87.349,-177.004,11.144,149.478
C04269=1111.784,369.029,-87.385,-177.000,11.146,149.478
C04270=1111.781,369.276,-87.422,-176.997,11.149,149.477
C04271=1111.777,369.523,-87.458,-176.994,11.151,149.477
C04272=1111.773,369.770,-87.495,-176.990,11.154,149.477
C04273=1111.770,370.018,-87.532,-176.987,11.156,149.477
C04274=1111.766,370.265,-87.569,-176.984,11.159,149.476
C04275=1111.762,370.512,-87.606,-176.980,11.161,149.476
C04276=1111.758,370.759,-87.642,-176.977,11.163,149.476
C04277=1111.755,371.007,-87.679,-176.974,11.166,149.476
C04278=1111.751,371.254,-87.716,-176.970,11.168,149.475
C04279=1111.747,371.501,-87.753,-176.967,11.171,149.475
C04280=1111.743,371.748,-87.789,-176.964,11.173,149.475
C04281=1111.739,371.995,-87.826,-176.960,11.176,149.475
C04282=1111.736,372.243,-87.864,-176.957,11.178,149.475
C04283=1111.732,372.490,-87.901,-176.954,11.181,149.474
C04284=1111.729,372.737,-87.937,-176.950,11.183,149.474
C04285=1111.725,372.984,-87.974,-176.947,11.185,149.474
C04286=1111.721,373.232,-88.011,-176.943,11.188,149.474
C04287=1111.717,373.479,-88.048,-176.940,11.190,149.473
C04288=1111.713,373.726,-88.085,-176.937,11.193,149.473
C04289=1111.710,373.973,-88.122,-176.934,11.195,149.473
C04290=1111.706,374.220,-88.159,-176.930,11.198,149.473
C04291=1111.702,374.467,-88.196,-176.927,11.200,149.473
C04292=1111.699,374.715,-88.233,-176.924,11.203,149.472
C04293=1111.695,374.962,-88.271,-176.920,11.205,149.472
C04294=1111.691,375.174,-88.302,-176.918,11.207,149.472
C04295=1111.689,375.386,-88.334,-176.915,11.210,149.472
C04296=1111.685,375.597,-88.365,-176.912,11.212,149.472
C04297=1111.682,375.808,-88.397,-176.909,11.214,149.472
C04298=1111.679,376.020,-88.429,-176.907,11.216,149.471
C04299=1111.676,376.232,-88.460,-176.903,11.219,149.471
C04300=1111.672,376.443,-88.492,-176.901,11.220,149.471
C04301=1111.669,376.655,-88.525,-176.898,11.223,149.471
C04302=1111.666,376.902,-88.562,-176.894,11.225,149.471
C04303=1111.662,377.150,-88.599,-176.891,11.228,149.471
C04304=1111.659,377.396,-88.636,-176.888,11.230,149.470
C04305=1111.655,377.643,-88.673,-176.885,11.233,149.470
C04306=1111.651,377.891,-88.711,-176.881,11.235,149.470
C04307=1111.647,378.138,-88.748,-176.878,11.238,149.470
C04308=1111.643,378.385,-88.785,-176.875,11.240,149.470
C04309=1111.640,378.632,-88.823,-176.872,11.243,149.470
C04310=1111.636,378.879,-88.860,-176.869,11.246,149.469
C04311=1111.633,379.127,-88.898,-176.865,11.249,149.469
C04312=1111.629,379.374,-88.935,-176.861,11.251,149.469
C04313=1111.625,379.620,-88.972,-176.858,11.254,149.469
C04314=1111.621,379.868,-89.009,-176.855,11.257,149.469
C04315=1111.617,380.115,-89.047,-176.852,11.259,149.469
C04316=1111.614,380.363,-89.085,-176.849,11.262,149.468
C04317=1111.609,380.610,-89.122,-176.845,11.264,149.468
C04318=1111.606,380.857,-89.160,-176.842,11.267,149.468
C04319=1111.602,381.104,-89.197,-176.839,11.270,149.468
C04320=1111.598,381.351,-89.235,-176.835,11.273,149.468
C04321=1111.595,381.598,-89.273,-176.832,11.275,149.468
C04322=1111.591,381.845,-89.309,-176.829,11.278,149.468
C04323=1111.588,382.092,-89.347,-176.826,11.281,149.467
C04324=1111.584,382.339,-89.385,-176.822,11.283,149.467
C04325=1111.580,382.587,-89.424,-176.819,11.286,149.467
C04326=1111.576,382.834,-89.460,-176.816,11.288,149.467
C04327=1111.573,383.081,-89.498,-176.813,11.292,149.467
C04328=1111.569,383.328,-89.536,-176.809,11.294,149.467
C04329=1111.566,383.575,-89.574,-176.806,11.297,149.467
C04330=1111.562,383.822,-89.611,-176.804,11.299,149.467
C04331=1111.558,384.070,-89.649,-176.801,11.302,149.467
C04332=1111.554,384.316,-89.687,-176.798,11.305,149.467
C04333=1111.551,384.564,-89.725,-176.796,11.307,149.467
C04334=1111.547,384.810,-89.762,-176.793,11.309,149.467
C04335=1111.544,385.057,-89.800,-176.790,11.312,149.467
C04336=1111.540,385.306,-89.838,-176.788,11.314,149.467
C04337=1111.536,385.552,-89.876,-176.785,11.317,149.467
C04338=1111.533,385.799,-89.914,-176.782,11.320,149.467
C04339=1111.529,386.046,-89.951,-176.779,11.323,149.467
C04340=1111.525,386.294,-89.990,-176.777,11.325,149.467
C04341=1111.521,386.540,-90.027,-176.774,11.328,149.467
C04342=1111.518,386.787,-90.065,-176.771,11.331,149.467
C04343=1111.514,387.034,-90.103,-176.769,11.334,149.467
C04344=1111.510,387.282,-90.141,-176.766,11.337,149.467
C04345=1111.507,387.529,-90.179,-176.764,11.339,149.467
C04346=1111.503,387.775,-90.217,-176.761,11.342,149.467
C04347=1111.500,388.023,-90.255,-176.758,11.345,149.467
C04348=1111.496,388.270,-90.293,-176.756,11.348,149.467
C04349=1111.493,388.517,-90.331,-176.753,11.351,149.467
C04350=1111.489,388.729,-90.364,-176.751,11.353,149.467
C04351=1111.486,388.940,-90.396,-176.748,11.356,149.467
C04352=1111.484,389.151,-90.429,-176.746,11.358,149.467
C04353=1111.480,389.362,-90.461,-176.744,11.361,149.468
C04354=1111.477,389.574,-90.493,-176.741,11.363,149.468
C04355=1111.474,389.786,-90.527,-176.740,11.366,149.468
C04356=1111.471,389.997,-90.559,-176.737,11.369,149.468
C04357=1111.468,390.208,-90.592,-176.735,11.371,149.468
C04358=1111.464,390.455,-90.630,-176.732,11.374,149.468
C04359=1111.460,390.703,-90.668,-176.730,11.377,149.468
C04360=1111.457,390.950,-90.706,-176.727,11.380,149.468
C04361=1111.453,391.196,-90.744,-176.725,11.384,149.469
C04362=1111.449,391.444,-90.783,-176.722,11.387,149.469
C04363=1111.446,391.691,-90.821,-176.719,11.391,149.469
C04364=1111.442,391.938,-90.859,-176.717,11.394,149.469
C04365=1111.439,392.185,-90.897,-176.714,11.397,149.469
C04366=1111.435,392.432,-90.935,-176.712,11.400,149.470
C04367=1111.432,392.679,-90.974,-176.710,11.404,149.470
C04368=1111.428,392.926,-91.012,-176.707,11.407,149.470
C04369=1111.424,393.173,-91.051,-176.704,11.411,149.470
C04370=1111.421,393.420,-91.089,-176.701,11.414,149.470
C04371=1111.417,393.667,-91.127,-176.699,11.417,149.471
C04372=1111.413,393.914,-91.165,-176.697,11.420,149.471
C04373=1111.410,394.161,-91.205,-176.694,11.425,149.471
C04374=1111.406,394.408,-91.242,-176.692,11.428,149.472
C04375=1111.402,394.655,-91.281,-176.690,11.431,149.472
C04376=1111.398,394.902,-91.320,-176.686,11.435,149.472
C04377=1111.395,395.149,-91.358,-176.684,11.439,149.473
C04378=1111.391,395.396,-91.397,-176.682,11.442,149.473
C04379=1111.388,395.643,-91.435,-176.679,11.446,149.473
C04380=1111.384,395.890,-91.474,-176.677,11.450,149.474
C04381=1111.381,396.137,-91.512,-176.675,11.453,149.474
C04382=1111.377,396.383,-91.551,-176.672,11.457,149.474
C04383=1111.373,396.631,-91.589,-176.670,11.460,149.475
C04384=1111.370,396.878,-91.628,-176.667,11.465,149.475
C04385=1111.366,397.125,-91.667,-176.665,11.468,149.475
C04386=1111.363,397.372,-91.705,-176.662,11.472,149.476
C04387=1111.359,397.619,-91.743,-176.660,11.476,149.476
C04388=1111.355,397.866,-91.783,-176.657,11.480,149.477
C04389=1111.352,398.112,-91.821,-176.655,11.484,149.477
C04390=1111.348,398.360,-91.860,-176.653,11.488,149.478
C04391=1111.345,398.607,-91.899,-176.651,11.492,149.478
C04392=1111.341,398.853,-91.937,-176.648,11.496,149.478
C04393=1111.337,399.100,-91.976,-176.646,11.501,149.479
C04394=1111.334,399.347,-92.015,-176.643,11.504,149.479
C04395=1111.330,399.595,-92.053,-176.641,11.509,149.480
C04396=1111.327,399.842,-92.092,-176.638,11.513,149.480
C04397=1111.323,400.089,-92.132,-176.637,11.517,149.481
C04398=1111.320,400.335,-92.170,-176.634,11.521,149.481
C04399=1111.316,400.582,-92.208,-176.632,11.525,149.482
C04400=1111.312,400.829,-92.248,-176.629,11.530,149.483
C04401=1111.309,401.076,-92.287,-176.628,11.534,149.483
C04402=1111.306,401.323,-92.326,-176.625,11.538,149.484
C04403=1111.302,401.570,-92.365,-176.622,11.543,149.484
C04404=1111.298,401.817,-92.403,-176.620,11.547,149.485
C04405=1111.295,402.064,-92.443,-176.618,11.552,149.485
C04406=1111.292,402.274,-92.476,-176.616,11.556,149.486
C04407=1111.289,402.486,-92.509,-176.614,11.559,149.486
C04408=1111.285,402.698,-92.542,-176.612,11.563,149.487
C04409=1111.283,402.909,-92.576,-176.610,11.567,149.487
C04410=1111.279,403.120,-92.610,-176.608,11.571,149.488
C04411=1111.276,403.332,-92.643,-176.606,11.575,149.489
C04412=1111.274,403.542,-92.676,-176.605,11.579,149.489
C04413=1111.270,403.754,-92.709,-176.603,11.583,149.490
C04414=1111.267,404.001,-92.748,-176.601,11.588,149.490
C04415=1111.263,404.248,-92.788,-176.599,11.592,149.491
C04416=1111.259,404.495,-92.827,-176.597,11.597,149.492
C04417=1111.256,404.742,-92.866,-176.594,11.602,149.493
C04418=1111.252,404.989,-92.905,-176.592,11.607,149.493
C04419=1111.249,405.235,-92.944,-176.589,11.612,149.494
C04420=1111.246,405.482,-92.983,-176.587,11.617,149.495
C04421=1111.242,405.729,-93.023,-176.585,11.622,149.495
C04422=1111.239,405.976,-93.062,-176.584,11.627,149.496
C04423=1111.235,406.223,-93.102,-176.582,11.632,149.497
C04424=1111.232,406.470,-93.141,-176.579,11.637,149.498
C04425=1111.228,406.717,-93.180,-176.577,11.642,149.499
C04426=1111.224,406.963,-93.220,-176.575,11.647,149.499
C04427=1111.221,407.210,-93.259,-176.573,11.652,149.500
C04428=1111.217,407.457,-93.298,-176.570,11.658,149.501
C04429=1111.214,407.704,-93.338,-176.569,11.663,149.502
C04430=1111.210,407.951,-93.377,-176.567,11.668,149.503
C04431=1111.207,408.198,-93.417,-176.564,11.673,149.504
C04432=1111.203,408.445,-93.456,-176.563,11.679,149.505
C04433=1111.199,408.692,-93.495,-176.561,11.684,149.505
C04434=1111.196,408.938,-93.535,-176.559,11.690,149.507
C04435=1111.192,409.185,-93.574,-176.557,11.695,149.507
C04436=1111.189,409.432,-93.614,-176.554,11.700,149.508
C04437=1111.185,409.678,-93.653,-176.553,11.706,149.509
C04438=1111.182,409.926,-93.693,-176.551,11.712,149.510
C04439=1111.179,410.173,-93.732,-176.549,11.717,149.511
C04440=1111.176,410.419,-93.772,-176.547,11.723,149.512
C04441=1111.172,410.666,-93.812,-176.545,11.728,149.513
C04442=1111.169,410.912,-93.852,-176.543,11.734,149.514
C04443=1111.165,411.159,-93.891,-176.541,11.739,149.515
C04444=1111.161,411.406,-93.930,-176.539,11.745,149.516
C04445=1111.157,411.653,-93.971,-176.537,11.751,149.517
C04446=1111.154,411.900,-94.010,-176.536,11.757,149.518
C04447=1111.151,412.147,-94.050,-176.534,11.763,149.520
C04448=1111.147,412.394,-94.089,-176.532,11.769,149.521
C04449=1111.144,412.640,-94.129,-176.530,11.775,149.522
C04450=1111.140,412.887,-94.169,-176.528,11.781,149.523
C04451=1111.137,413.134,-94.209,-176.526,11.787,149.524
C04452=1111.133,413.380,-94.249,-176.524,11.793,149.525
C04453=1111.130,413.628,-94.289,-176.522,11.799,149.526
C04454=1111.128,413.875,-94.329,-176.521,11.806,149.528
C04455=1111.126,414.121,-94.368,-176.519,11.811,149.529
C04456=1111.124,414.368,-94.408,-176.518,11.818,149.530
C04457=1111.123,414.615,-94.447,-176.516,11.824,149.531
C04458=1111.122,414.862,-94.487,-176.514,11.830,149.532
C04459=1111.122,415.109,-94.526,-176.512,11.837,149.534
C04460=1111.123,415.355,-94.566,-176.511,11.843,149.535
C04461=1111.124,415.603,-94.605,-176.509,11.850,149.536
C04462=1111.125,415.814,-94.639,-176.508,11.855,149.537
C04463=1111.127,416.024,-94.672,-176.506,11.861,149.538
C04464=1111.129,416.235,-94.706,-176.505,11.866,149.540
C04465=1111.131,416.447,-94.739,-176.504,11.871,149.541
C04466=1111.133,416.658,-94.773,-176.502,11.877,149.542
C04467=1111.137,416.868,-94.806,-176.501,11.882,149.543
C04468=1111.140,417.080,-94.839,-176.499,11.889,149.544
C04469=1111.144,417.290,-94.872,-176.498,11.894,149.545
C04470=1110.725,417.290,-94.935,-176.491,11.899,149.545
C04471=1110.721,417.079,-94.903,-176.492,11.893,149.543
C04472=1110.718,416.868,-94.869,-176.493,11.888,149.542
C04473=1110.714,416.658,-94.835,-176.495,11.881,149.541
C04474=1110.712,416.447,-94.802,-176.497,11.876,149.540
C04475=1110.710,416.235,-94.769,-176.498,11.871,149.539
C04476=1110.708,416.024,-94.735,-176.499,11.865,149.538
C04477=1110.706,415.814,-94.701,-176.500,11.859,149.537
C04478=1110.705,415.602,-94.667,-176.502,11.854,149.536
C04479=1110.704,415.355,-94.628,-176.503,11.848,149.534
C04480=1110.703,415.108,-94.588,-176.505,11.841,149.533
C04481=1110.703,414.862,-94.549,-176.507,11.835,149.532
C04482=1110.704,414.615,-94.510,-176.509,11.829,149.531
C04483=1110.705,414.367,-94.470,-176.510,11.822,149.529
C04484=1110.707,414.121,-94.431,-176.512,11.816,149.528
C04485=1110.709,413.874,-94.391,-176.514,11.810,149.527
C04486=1110.711,413.627,-94.351,-176.516,11.803,149.526
C04487=1110.714,413.381,-94.311,-176.518,11.797,149.525
C04488=1110.718,413.134,-94.271,-176.520,11.791,149.523
C04489=1110.721,412.887,-94.231,-176.522,11.785,149.522
C04490=1110.724,412.640,-94.191,-176.524,11.778,149.521
C04491=1110.728,412.393,-94.152,-176.525,11.773,149.520
C04492=1110.731,412.147,-94.112,-176.527,11.767,149.519
C04493=1110.735,411.900,-94.073,-176.530,11.761,149.518
C04494=1110.739,411.653,-94.032,-176.531,11.754,149.517
C04495=1110.742,411.406,-93.993,-176.533,11.749,149.516
C04496=1110.746,411.160,-93.953,-176.535,11.743,149.515
C04497=1110.749,410.912,-93.913,-176.537,11.737,149.514
C04498=1110.752,410.666,-93.873,-176.539,11.732,149.513
C04499=1110.756,410.419,-93.834,-176.541,11.726,149.512
C04500=1110.759,410.172,-93.795,-176.543,11.720,149.511
C04501=1110.763,409.926,-93.755,-176.545,11.715,149.510
C04502=1110.766,409.679,-93.716,-176.547,11.709,149.509
C04503=1110.770,409.432,-93.676,-176.549,11.704,149.508
C04504=1110.774,409.185,-93.636,-176.551,11.698,149.507
C04505=1110.777,408.938,-93.596,-176.553,11.693,149.506
C04506=1110.781,408.691,-93.557,-176.555,11.687,149.505
C04507=1110.784,408.444,-93.517,-176.557,11.682,149.504
C04508=1110.787,408.197,-93.478,-176.560,11.676,149.503
C04509=1110.791,407.950,-93.438,-176.562,11.671,149.502
C04510=1110.795,407.703,-93.399,-176.563,11.666,149.501
C04511=1110.798,407.457,-93.359,-176.566,11.660,149.501
C04512=1110.802,407.210,-93.320,-176.568,11.655,149.500
C04513=1110.805,406.963,-93.281,-176.570,11.650,149.499
C04514=1110.808,406.716,-93.242,-176.572,11.645,149.498
C04515=1110.812,406.469,-93.203,-176.574,11.640,149.497
C04516=1110.815,406.223,-93.163,-176.576,11.635,149.497
C04517=1110.819,405.976,-93.124,-176.579,11.629,149.496
C04518=1110.822,405.729,-93.084,-176.581,11.624,149.495
C04519=1110.826,405.482,-93.045,-176.583,11.619,149.494
C04520=1110.830,405.235,-93.006,-176.585,11.615,149.494
C04521=1110.833,404.988,-92.967,-176.587,11.610,149.493
C04522=1110.837,404.741,-92.927,-176.589,11.605,149.492
C04523=1110.840,404.494,-92.888,-176.592,11.600,149.491
C04524=1110.844,404.247,-92.849,-176.594,11.595,149.491
C04525=1110.847,404.001,-92.810,-176.596,11.590,149.490
C04526=1110.850,403.754,-92.771,-176.599,11.586,149.489
C04527=1110.854,403.543,-92.738,-176.600,11.582,149.489
C04528=1110.857,403.332,-92.704,-176.602,11.578,149.488
C04529=1110.860,403.120,-92.671,-176.604,11.573,149.488
C04530=1110.863,402.909,-92.637,-176.606,11.570,149.487
C04531=1110.866,402.698,-92.604,-176.608,11.566,149.487
C04532=1110.868,402.486,-92.570,-176.610,11.562,149.486
C04533=1110.872,402.275,-92.537,-176.612,11.558,149.486
C04534=1110.875,402.064,-92.504,-176.614,11.554,149.485
C04535=1110.879,401.817,-92.464,-176.616,11.549,149.484
C04536=1110.882,401.570,-92.426,-176.619,11.545,149.484
C04537=1110.886,401.323,-92.386,-176.621,11.540,149.483
C04538=1110.889,401.076,-92.347,-176.623,11.536,149.483
C04539=1110.893,400.829,-92.309,-176.626,11.532,149.482
C04540=1110.897,400.583,-92.270,-176.628,11.528,149.482
C04541=1110.900,400.336,-92.231,-176.630,11.523,149.481
C04542=1110.904,400.089,-92.192,-176.633,11.519,149.481
C04543=1110.908,399.841,-92.153,-176.635,11.515,149.480
C04544=1110.911,399.595,-92.115,-176.637,11.511,149.480
C04545=1110.914,399.348,-92.075,-176.640,11.506,149.479
C04546=1110.918,399.101,-92.036,-176.642,11.503,149.479
C04547=1110.922,398.854,-91.999,-176.645,11.498,149.478
C04548=1110.925,398.607,-91.959,-176.647,11.494,149.478
C04549=1110.929,398.360,-91.920,-176.649,11.490,149.477
C04550=1110.932,398.113,-91.882,-176.652,11.486,149.477
C04551=1110.936,397.866,-91.843,-176.655,11.482,149.476
C04552=1110.940,397.619,-91.805,-176.657,11.478,149.476
C04553=1110.943,397.372,-91.766,-176.659,11.474,149.476
C04554=1110.947,397.125,-91.727,-176.661,11.471,149.475
C04555=1110.951,396.878,-91.688,-176.664,11.466,149.475
C04556=1110.953,396.631,-91.650,-176.666,11.463,149.474
C04557=1110.958,396.384,-91.612,-176.669,11.459,149.474
C04558=1110.961,396.138,-91.573,-176.671,11.455,149.474
C04559=1110.965,395.890,-91.534,-176.674,11.451,149.473
C04560=1110.968,395.643,-91.495,-176.676,11.448,149.473
C04561=1110.972,395.397,-91.458,-176.679,11.444,149.473
C04562=1110.976,395.150,-91.418,-176.681,11.440,149.472
C04563=1110.979,394.902,-91.380,-176.684,11.437,149.472
C04564=1110.983,394.655,-91.342,-176.686,11.433,149.472
C04565=1110.986,394.409,-91.303,-176.689,11.430,149.471
C04566=1110.990,394.161,-91.265,-176.692,11.425,149.471
C04567=1110.993,393.915,-91.226,-176.694,11.422,149.471
C04568=1110.997,393.667,-91.188,-176.697,11.419,149.471
C04569=1111.001,393.420,-91.150,-176.699,11.415,149.470
C04570=1111.005,393.173,-91.111,-176.702,11.412,149.470
C04571=1111.008,392.926,-91.073,-176.704,11.408,149.470
C04572=1111.012,392.679,-91.035,-176.707,11.405,149.470
C04573=1111.015,392.433,-90.996,-176.709,11.402,149.469
C04574=1111.019,392.185,-90.958,-176.712,11.398,149.469
C04575=1111.023,391.938,-90.920,-176.715,11.395,149.469
C04576=1111.027,391.691,-90.882,-176.717,11.392,149.469
C04577=1111.030,391.444,-90.843,-176.720,11.388,149.469
C04578=1111.034,391.197,-90.804,-176.722,11.385,149.468
C04579=1111.037,390.950,-90.767,-176.725,11.382,149.468
C04580=1111.041,390.703,-90.729,-176.728,11.379,149.468
C04581=1111.045,390.455,-90.690,-176.731,11.375,149.468
C04582=1111.048,390.209,-90.652,-176.733,11.372,149.468
C04583=1111.051,389.997,-90.619,-176.735,11.370,149.468
C04584=1111.055,389.786,-90.587,-176.738,11.367,149.468
C04585=1111.057,389.575,-90.554,-176.740,11.365,149.467
C04586=1111.060,389.362,-90.522,-176.742,11.362,149.467
C04587=1111.063,389.152,-90.489,-176.744,11.359,149.467
C04588=1111.067,388.940,-90.456,-176.746,11.357,149.467
C04589=1111.070,388.729,-90.424,-176.749,11.354,149.467
C04590=1111.073,388.517,-90.391,-176.751,11.352,149.467
C04591=1111.077,388.271,-90.354,-176.754,11.349,149.467
C04592=1111.080,388.023,-90.316,-176.757,11.346,149.467
C04593=1111.084,387.776,-90.277,-176.759,11.343,149.467
C04594=1111.088,387.529,-90.240,-176.762,11.340,149.467
C04595=1111.091,387.282,-90.202,-176.765,11.337,149.467
C04596=1111.096,387.035,-90.163,-176.767,11.334,149.467
C04597=1111.099,386.788,-90.126,-176.770,11.332,149.467
C04598=1111.102,386.540,-90.088,-176.773,11.329,149.467
C04599=1111.106,386.294,-90.050,-176.775,11.326,149.467
C04600=1111.110,386.046,-90.011,-176.778,11.323,149.466
C04601=1111.113,385.800,-89.974,-176.781,11.320,149.466
C04602=1111.117,385.552,-89.936,-176.783,11.318,149.466
C04603=1111.120,385.306,-89.898,-176.786,11.316,149.466
C04604=1111.124,385.058,-89.860,-176.789,11.313,149.466
C04605=1111.127,384.811,-89.822,-176.792,11.310,149.466
C04606=1111.131,384.564,-89.784,-176.794,11.308,149.467
C04607=1111.135,384.317,-89.747,-176.797,11.305,149.467
C04608=1111.139,384.070,-89.710,-176.800,11.302,149.467
C04609=1111.142,383.822,-89.671,-176.803,11.300,149.467
C04610=1111.146,383.576,-89.633,-176.805,11.298,149.467
C04611=1111.149,383.329,-89.596,-176.808,11.295,149.467
C04612=1111.154,383.081,-89.559,-176.812,11.292,149.467
C04613=1111.157,382.834,-89.521,-176.815,11.290,149.467
C04614=1111.161,382.587,-89.483,-176.818,11.286,149.467
C04615=1111.164,382.340,-89.445,-176.822,11.284,149.467
C04616=1111.169,382.093,-89.408,-176.825,11.281,149.467
C04617=1111.172,381.845,-89.370,-176.828,11.279,149.468
C04618=1111.176,381.599,-89.332,-176.831,11.276,149.468
C04619=1111.179,381.351,-89.295,-176.834,11.273,149.468
C04620=1111.183,381.104,-89.257,-176.838,11.270,149.468
C04621=1111.187,380.858,-89.220,-176.841,11.267,149.468
C04622=1111.190,380.610,-89.183,-176.845,11.265,149.468
C04623=1111.194,380.363,-89.145,-176.847,11.262,149.468
C04624=1111.197,380.115,-89.108,-176.851,11.260,149.468
C04625=1111.201,379.869,-89.070,-176.854,11.257,149.469
C04626=1111.204,379.622,-89.032,-176.857,11.255,149.469
C04627=1111.209,379.374,-88.995,-176.860,11.252,149.469
C04628=1111.213,379.128,-88.957,-176.864,11.249,149.469
C04629=1111.216,378.880,-88.920,-176.867,11.246,149.469
C04630=1111.220,378.633,-88.883,-176.871,11.244,149.469
C04631=1111.224,378.385,-88.845,-176.874,11.241,149.470
C04632=1111.228,378.139,-88.808,-176.877,11.239,149.470
C04633=1111.232,377.891,-88.771,-176.881,11.236,149.470
C04634=1111.235,377.644,-88.733,-176.884,11.233,149.470
C04635=1111.239,377.397,-88.696,-176.887,11.231,149.470
C04636=1111.242,377.150,-88.660,-176.890,11.228,149.470
C04637=1111.245,376.903,-88.622,-176.893,11.226,149.471
C04638=1111.250,376.656,-88.585,-176.897,11.223,149.471
C04639=1111.253,376.443,-88.552,-176.900,11.221,149.471
C04640=1111.256,376.232,-88.521,-176.902,11.219,149.471
C04641=1111.260,376.021,-88.489,-176.906,11.216,149.471
C04642=1111.262,375.809,-88.457,-176.908,11.215,149.472
C04643=1111.266,375.597,-88.426,-176.912,11.212,149.472
C04644=1111.269,375.386,-88.394,-176.914,11.210,149.472
C04645=1111.272,375.174,-88.362,-176.917,11.208,149.472
C04646=1111.275,374.963,-88.330,-176.920,11.206,149.472
C04647=1111.279,374.716,-88.293,-176.923,11.204,149.472
C04648=1111.282,374.468,-88.255,-176.926,11.201,149.473
C04649=1111.287,374.221,-88.219,-176.930,11.199,149.473
C04650=1111.290,373.974,-88.182,-176.933,11.196,149.473
C04651=1111.294,373.727,-88.146,-176.936,11.194,149.473
C04652=1111.297,373.479,-88.108,-176.940,11.191,149.473
C04653=1111.301,373.233,-88.071,-176.943,11.188,149.474
C04654=1111.305,372.985,-88.034,-176.947,11.185,149.474
C04655=1111.309,372.737,-87.997,-176.950,11.183,149.474
C04656=1111.312,372.491,-87.960,-176.953,11.180,149.474
C04657=1111.316,372.243,-87.924,-176.957,11.178,149.474
C04658=1111.320,371.996,-87.887,-176.960,11.176,149.475
C04659=1111.324,371.748,-87.849,-176.963,11.173,149.475
C04660=1111.327,371.501,-87.813,-176.967,11.171,149.475
C04661=1111.331,371.254,-87.776,-176.970,11.168,149.475
C04662=1111.335,371.007,-87.739,-176.974,11.166,149.476
C04663=1111.339,370.760,-87.702,-176.977,11.163,149.476
C04664=1111.342,370.513,-87.665,-176.980,11.161,149.476
C04665=1111.346,370.266,-87.628,-176.983,11.159,149.476
C04666=1111.350,370.018,-87.592,-176.987,11.156,149.476
C04667=1111.354,369.771,-87.556,-176.990,11.154,149.477
C04668=1111.357,369.523,-87.519,-176.993,11.151,149.477
C04669=1111.361,369.276,-87.482,-176.997,11.149,149.477
C04670=1111.365,369.029,-87.446,-177.000,11.146,149.478
C04671=1111.369,368.782,-87.409,-177.004,11.144,149.478
C04672=1111.373,368.535,-87.372,-177.007,11.141,149.478
C04673=1111.376,368.287,-87.335,-177.010,11.139,149.478
C04674=1111.380,368.040,-87.298,-177.014,11.137,149.478
C04675=1111.384,367.793,-87.262,-177.017,11.134,149.479
C04676=1111.388,367.545,-87.226,-177.021,11.132,149.479
C04677=1111.392,367.298,-87.189,-177.024,11.129,149.479
C04678=1111.395,367.051,-87.153,-177.027,11.127,149.479
C04679=1111.399,366.804,-87.116,-177.030,11.124,149.480
C04680=1111.403,366.556,-87.079,-177.034,11.122,149.480
C04681=1111.406,366.309,-87.043,-177.037,11.120,149.480
C04682=1111.410,366.061,-87.006,-177.041,11.117,149.480
C04683=1111.414,365.814,-86.970,-177.044,11.115,149.481
C04684=1111.418,365.567,-86.933,-177.047,11.112,149.481
C04685=1111.421,365.320,-86.898,-177.051,11.110,149.481
C04686=1111.426,365.073,-86.861,-177.054,11.108,149.481
C04687=1111.429,364.826,-86.825,-177.058,11.105,149.482
C04688=1111.433,364.578,-86.788,-177.061,11.103,149.482
C04689=1111.437,364.331,-86.752,-177.064,11.100,149.482
C04690=1111.441,364.082,-86.716,-177.067,11.099,149.482
C04691=1111.444,363.836,-86.679,-177.071,11.097,149.483
C04692=1111.448,363.588,-86.643,-177.074,11.094,149.483
C04693=1111.452,363.341,-86.607,-177.077,11.092,149.483
C04694=1111.456,363.094,-86.570,-177.081,11.089,149.484
C04695=1111.459,362.882,-86.540,-177.084,11.087,149.484
C04696=1111.462,362.670,-86.509,-177.087,11.085,149.484
C04697=1111.466,362.459,-86.477,-177.090,11.083,149.484
C04698=1111.469,362.247,-86.447,-177.093,11.081,149.484
C04699=1111.472,362.035,-86.416,-177.095,11.079,149.485
C04700=1111.475,361.823,-86.384,-177.098,11.077,149.485
C04701=1111.478,361.612,-86.354,-177.101,11.075,149.485
C04702=1111.481,361.400,-86.323,-177.104,11.073,149.485
C04703=1111.485,361.153,-86.287,-177.108,11.070,149.485
C04704=1111.489,360.905,-86.250,-177.111,11.068,149.486
C04705=1111.493,360.657,-86.215,-177.114,11.065,149.486
C04706=1111.496,360.411,-86.179,-177.118,11.063,149.486
C04707=1111.501,360.163,-86.143,-177.121,11.060,149.486
C04708=1111.504,359.916,-86.106,-177.124,11.059,149.487
C04709=1111.508,359.668,-86.071,-177.127,11.056,149.487
C04710=1111.511,359.421,-86.035,-177.131,11.054,149.487
C04711=1111.515,359.174,-85.998,-177.134,11.052,149.488
C04712=1111.519,358.926,-85.963,-177.138,11.049,149.488
C04713=1111.523,358.679,-85.927,-177.141,11.047,149.488
C04714=1111.527,358.431,-85.891,-177.144,11.044,149.488
C04715=1111.530,358.184,-85.855,-177.148,11.042,149.488
C04716=1111.534,357.937,-85.819,-177.151,11.039,149.489
C04717=1111.538,357.689,-85.784,-177.155,11.037,149.489
C04718=1111.542,357.441,-85.748,-177.158,11.035,149.489
C04719=1111.546,357.194,-85.711,-177.161,11.032,149.489
C04720=1111.550,356.948,-85.676,-177.165,11.030,149.490
C04721=1111.553,356.700,-85.641,-177.168,11.027,149.490
C04722=1111.557,356.453,-85.605,-177.171,11.025,149.490
C04723=1111.562,356.205,-85.569,-177.175,11.023,149.491
C04724=1111.565,355.957,-85.533,-177.178,11.020,149.491
C04725=1111.569,355.710,-85.497,-177.181,11.018,149.491
C04726=1111.572,355.463,-85.462,-177.185,11.015,149.491
C04727=1111.576,355.215,-85.426,-177.188,11.013,149.491
C04728=1111.580,354.968,-85.390,-177.191,11.010,149.492
C04729=1111.584,354.720,-85.354,-177.195,11.008,149.492
C04730=1111.588,354.473,-85.319,-177.198,11.006,149.492
C04731=1111.592,354.226,-85.284,-177.202,11.003,149.493
C04732=1111.596,353.978,-85.248,-177.205,11.001,149.493
C04733=1111.599,353.731,-85.212,-177.208,10.998,149.493
C04734=1111.603,353.483,-85.177,-177.212,10.996,149.493
C04735=1111.607,353.236,-85.141,-177.215,10.994,149.493
C04736=1111.611,352.989,-85.106,-177.218,10.991,149.494
C04737=1111.614,352.741,-85.071,-177.222,10.989,149.494
C04738=1111.619,352.494,-85.035,-177.225,10.986,149.494
C04739=1111.623,352.246,-84.999,-177.228,10.984,149.494
C04740=1111.626,351.999,-84.963,-177.231,10.981,149.495
C04741=1111.630,351.751,-84.929,-177.235,10.979,149.495
C04742=1111.634,351.504,-84.893,-177.238,10.976,149.495
C04743=1111.638,351.256,-84.858,-177.241,10.974,149.495
C04744=1111.642,351.009,-84.822,-177.245,10.971,149.495
C04745=1111.645,350.761,-84.787,-177.248,10.969,149.496
C04746=1111.650,350.514,-84.752,-177.251,10.966,149.496
C04747=1111.654,350.266,-84.717,-177.255,10.964,149.496
C04748=1111.657,350.019,-84.681,-177.258,10.962,149.496
C04749=1111.661,349.771,-84.646,-177.261,10.959,149.497
C04750=1111.665,349.525,-84.610,-177.265,10.956,149.497
C04751=1111.668,349.312,-84.581,-177.268,10.954,149.497
C04752=1111.671,349.101,-84.551,-177.270,10.952,149.497
C04753=1111.675,348.888,-84.520,-177.273,10.950,149.497
C04754=1111.678,348.676,-84.490,-177.276,10.948,149.498
C04755=1111.681,348.465,-84.460,-177.278,10.946,149.498
C04756=1111.684,348.253,-84.430,-177.282,10.943,149.498
C04757=1111.688,348.041,-84.399,-177.284,10.941,149.498
C04758=1111.691,347.828,-84.370,-177.287,10.940,149.498
C04759=1111.695,347.582,-84.334,-177.290,10.937,149.498
C04760=1111.699,347.333,-84.300,-177.293,10.935,149.499
C04761=1111.703,347.086,-84.264,-177.296,10.932,149.499
C04762=1111.707,346.839,-84.229,-177.300,10.930,149.499
C04763=1111.711,346.591,-84.195,-177.303,10.927,149.499
C04764=1111.714,346.344,-84.159,-177.306,10.925,149.499
C04765=1111.719,346.096,-84.125,-177.310,10.922,149.500
C04766=1111.722,345.849,-84.089,-177.312,10.920,149.500
C04767=1111.726,345.601,-84.054,-177.315,10.918,149.500
C04768=1111.731,345.354,-84.019,-177.318,10.915,149.500
C04769=1111.734,345.106,-83.985,-177.322,10.913,149.500
C04770=1111.738,344.859,-83.949,-177.325,10.910,149.501
C04771=1111.742,344.611,-83.915,-177.328,10.908,149.501
C04772=1111.746,344.364,-83.879,-177.331,10.905,149.501
C04773=1111.750,344.116,-83.844,-177.335,10.903,149.501
C04774=1111.754,343.869,-83.811,-177.338,10.900,149.501
C04775=1111.757,343.621,-83.775,-177.341,10.898,149.502
C04776=1111.762,343.374,-83.741,-177.344,10.896,149.502
C04777=1111.766,343.126,-83.705,-177.347,10.893,149.502
C04778=1111.769,342.878,-83.671,-177.350,10.891,149.502
C04779=1111.773,342.631,-83.636,-177.353,10.888,149.502
C04780=1111.777,342.383,-83.601,-177.357,10.886,149.503
C04781=1111.782,342.136,-83.566,-177.360,10.883,149.503
C04782=1111.785,341.888,-83.532,-177.363,10.881,149.503
C04783=1111.789,341.641,-83.497,-177.366,10.878,149.503
C04784=1111.793,341.393,-83.462,-177.370,10.876,149.503
C04785=1111.796,341.145,-83.428,-177.373,10.873,149.504
C04786=1111.801,340.898,-83.393,-177.376,10.871,149.504
C04787=1111.804,340.650,-83.358,-177.379,10.869,149.504
C04788=1111.808,340.403,-83.324,-177.382,10.866,149.504
C04789=1111.812,340.155,-83.289,-177.385,10.864,149.504
C04790=1111.817,339.908,-83.255,-177.388,10.861,149.504
C04791=1111.820,339.660,-83.220,-177.391,10.859,149.505
C04792=1111.825,339.413,-83.186,-177.395,10.856,149.505
C04793=1111.828,339.165,-83.150,-177.398,10.854,149.505
C04794=1111.832,338.918,-83.116,-177.401,10.851,149.505
C04795=1111.836,338.670,-83.082,-177.404,10.849,149.505
C04796=1111.840,338.423,-83.048,-177.408,10.846,149.506
C04797=1111.844,338.175,-83.013,-177.410,10.844,149.506
C04798=1111.848,337.927,-82.978,-177.414,10.842,149.506
C04799=1111.852,337.679,-82.944,-177.417,10.839,149.506
C04800=1111.856,337.432,-82.910,-177.420,10.837,149.506
C04801=1111.860,337.184,-82.876,-177.423,10.834,149.507
C04802=1111.864,336.937,-82.841,-177.426,10.832,149.507
C04803=1111.867,336.689,-82.807,-177.429,10.829,149.507
C04804=1111.872,336.442,-82.772,-177.433,10.827,149.507
C04805=1111.875,336.194,-82.738,-177.436,10.824,149.507
C04806=1111.880,335.946,-82.704,-177.439,10.821,149.507
C04807=1111.883,335.734,-82.674,-177.442,10.820,149.508
C04808=1111.886,335.523,-82.645,-177.444,10.818,149.508
C04809=1111.889,335.311,-82.616,-177.447,10.815,149.508
C04810=1111.892,335.098,-82.586,-177.450,10.813,149.508
C04811=1111.896,334.887,-82.557,-177.452,10.812,149.508
C04812=1111.900,334.674,-82.528,-177.455,10.809,149.508
C04813=1111.903,334.462,-82.499,-177.458,10.807,149.509
C04814=1111.907,334.250,-82.469,-177.460,10.805,149.509
C04815=1111.910,334.002,-82.435,-177.463,10.803,149.509
C04816=1111.914,333.755,-82.401,-177.467,10.800,149.509
C04817=1111.918,333.507,-82.366,-177.470,10.797,149.509
C04818=1111.922,333.260,-82.332,-177.473,10.795,149.510
C04819=1111.927,333.012,-82.299,-177.476,10.792,149.510
C04820=1111.930,332.764,-82.264,-177.480,10.790,149.510
C04821=1111.934,332.517,-82.231,-177.483,10.787,149.510
C04822=1111.938,332.269,-82.196,-177.486,10.785,149.510
C04823=1111.942,332.021,-82.163,-177.489,10.783,149.511
C04824=1111.946,331.774,-82.129,-177.491,10.780,149.511
C04825=1111.949,331.526,-82.094,-177.495,10.778,149.511
C04826=1111.954,331.278,-82.061,-177.498,10.775,149.511
C04827=1111.957,331.031,-82.027,-177.501,10.773,149.511
C04828=1111.961,330.783,-81.992,-177.504,10.770,149.511
C04829=1111.966,330.535,-81.959,-177.508,10.768,149.512
C04830=1111.969,330.288,-81.925,-177.511,10.765,149.512
C04831=1111.973,330.040,-81.891,-177.514,10.763,149.512
C04832=1111.977,329.792,-81.857,-177.517,10.760,149.512
C04833=1111.981,329.545,-81.823,-177.521,10.758,149.512
C04834=1111.985,329.297,-81.790,-177.523,10.756,149.513
C04835=1111.989,329.050,-81.756,-177.526,10.753,149.513
C04836=1111.993,328.802,-81.721,-177.529,10.751,149.513
C04837=1111.997,328.554,-81.688,-177.532,10.748,149.513
C04838=1112.001,328.307,-81.654,-177.536,10.745,149.513
C04839=1112.005,328.059,-81.621,-177.539,10.743,149.514
C04840=1112.009,327.812,-81.586,-177.542,10.740,149.514
C04841=1112.013,327.563,-81.553,-177.545,10.738,149.514
C04842=1112.017,327.316,-81.519,-177.549,10.735,149.514
C04843=1112.021,327.068,-81.486,-177.552,10.733,149.514
C04844=1112.025,326.821,-81.453,-177.554,10.731,149.514
C04845=1112.028,326.573,-81.418,-177.558,10.728,149.515
C04846=1112.033,326.325,-81.385,-177.560,10.726,149.515
C04847=1112.037,326.078,-81.351,-177.564,10.723,149.515
C04848=1112.041,325.830,-81.318,-177.567,10.721,149.515
C04849=1112.045,325.581,-81.284,-177.570,10.718,149.515
C04850=1112.048,325.334,-81.250,-177.573,10.716,149.516
C04851=1112.053,325.087,-81.217,-177.577,10.713,149.516
C04852=1112.057,324.839,-81.184,-177.580,10.710,149.516
C04853=1112.060,324.591,-81.150,-177.583,10.708,149.516
C04854=1112.064,324.343,-81.116,-177.586,10.706,149.516
C04855=1112.069,324.095,-81.083,-177.589,10.703,149.516
C04856=1112.073,323.848,-81.049,-177.592,10.701,149.517
C04857=1112.077,323.600,-81.016,-177.595,10.699,149.517
C04858=1112.080,323.352,-80.982,-177.598,10.696,149.517
C04859=1112.085,323.104,-80.949,-177.601,10.693,149.517
C04860=1112.088,322.857,-80.915,-177.605,10.691,149.517
C04861=1112.093,322.609,-80.882,-177.608,10.688,149.518
C04862=1112.097,322.362,-80.849,-177.611,10.686,149.518
C04863=1112.099,322.149,-80.821,-177.613,10.684,149.518
C04864=1112.104,321.937,-80.792,-177.616,10.682,149.518
C04865=1112.106,321.725,-80.763,-177.619,10.679,149.518
C04866=1112.110,321.513,-80.735,-177.621,10.677,149.518
C04867=1112.113,321.300,-80.706,-177.624,10.676,149.519
C04868=1112.116,321.088,-80.678,-177.627,10.673,149.519
C04869=1112.120,320.876,-80.650,-177.629,10.671,149.519
C04870=1112.123,320.664,-80.621,-177.632,10.669,149.519
C04871=1112.127,320.417,-80.588,-177.635,10.667,149.519
C04872=1112.131,320.169,-80.554,-177.638,10.664,149.519
C04873=1112.135,319.921,-80.521,-177.641,10.661,149.520
C04874=1112.140,319.673,-80.488,-177.644,10.659,149.520
C04875=1112.144,319.426,-80.455,-177.648,10.656,149.520
C04876=1112.147,319.177,-80.421,-177.651,10.654,149.520
C04877=1112.151,318.930,-80.388,-177.654,10.651,149.520
C04878=1112.155,318.682,-80.356,-177.657,10.649,149.520
C04879=1112.159,318.434,-80.323,-177.660,10.646,149.521
C04880=1112.163,318.187,-80.289,-177.663,10.644,149.521
C04881=1112.167,317.939,-80.256,-177.666,10.642,149.521
C04882=1112.172,317.691,-80.224,-177.669,10.639,149.521
C04883=1112.176,317.443,-80.191,-177.672,10.636,149.521
C04884=1112.179,317.195,-80.158,-177.676,10.634,149.522
C04885=1112.183,316.948,-80.125,-177.679,10.631,149.522
C04886=1112.187,316.700,-80.092,-177.682,10.629,149.522
C04887=1112.192,316.452,-80.059,-177.685,10.626,149.522
C04888=1112.196,316.205,-80.026,-177.688,10.624,149.522
C04889=1112.199,315.957,-79.993,-177.692,10.621,149.523
C04890=1112.204,315.709,-79.961,-177.694,10.619,149.523
C04891=1112.208,315.461,-79.927,-177.697,10.617,149.523
C04892=1112.212,315.213,-79.894,-177.700,10.614,149.523
C04893=1112.215,314.966,-79.862,-177.703,10.611,149.523
C04894=1112.220,314.718,-79.829,-177.706,10.609,149.523
C04895=1112.224,314.470,-79.796,-177.710,10.606,149.524
C04896=1112.228,314.222,-79.763,-177.713,10.604,149.524
C04897=1112.231,313.975,-79.730,-177.716,10.601,149.524
C04898=1112.236,313.726,-79.698,-177.719,10.599,149.524
C04899=1112.240,313.479,-79.665,-177.722,10.596,149.524
C04900=1112.243,313.231,-79.632,-177.725,10.594,149.524
C04901=1112.248,312.983,-79.600,-177.728,10.591,149.525
C04902=1112.252,312.735,-79.567,-177.731,10.589,149.525
C04903=1112.255,312.488,-79.534,-177.734,10.587,149.525
C04904=1112.260,312.239,-79.502,-177.737,10.584,149.525
C04905=1112.264,311.992,-79.468,-177.741,10.581,149.525
C04906=1112.268,311.744,-79.437,-177.744,10.579,149.525
C04907=1112.272,311.496,-79.403,-177.747,10.576,149.526
C04908=1112.275,311.248,-79.372,-177.750,10.573,149.526
C04909=1112.280,311.000,-79.338,-177.753,10.571,149.526
C04910=1112.284,310.752,-79.306,-177.756,10.569,149.526
C04911=1112.287,310.504,-79.273,-177.759,10.566,149.526
C04912=1112.292,310.256,-79.241,-177.762,10.564,149.527
C04913=1112.296,310.009,-79.209,-177.765,10.561,149.527
C04914=1112.300,309.761,-79.176,-177.768,10.559,149.527
C04915=1112.304,309.513,-79.143,-177.771,10.556,149.527
C04916=1112.308,309.265,-79.111,-177.775,10.554,149.527
C04917=1112.312,309.017,-79.078,-177.778,10.551,149.527
C04918=1112.316,308.769,-79.046,-177.781,10.548,149.528
C04919=1112.319,308.557,-79.018,-177.783,10.546,149.528
C04920=1112.323,308.345,-78.991,-177.786,10.545,149.528
C04921=1112.327,308.132,-78.962,-177.789,10.542,149.528
C04922=1112.330,307.920,-78.935,-177.791,10.540,149.528
C04923=1112.334,307.708,-78.907,-177.794,10.538,149.529
C04924=1112.337,307.495,-78.880,-177.797,10.536,149.529
C04925=1112.341,307.283,-78.852,-177.799,10.534,149.529
C04926=1112.344,307.070,-78.824,-177.802,10.532,149.529
C04927=1112.348,306.823,-78.793,-177.805,10.529,149.529
C04928=1112.352,306.575,-78.760,-177.808,10.527,149.529
C04929=1112.356,306.327,-78.728,-177.811,10.524,149.529
C04930=1112.360,306.079,-78.696,-177.814,10.521,149.530
C04931=1112.364,305.831,-78.663,-177.817,10.519,149.530
C04932=1112.369,305.584,-78.631,-177.821,10.516,149.530
C04933=1112.373,305.336,-78.599,-177.823,10.514,149.530
C04934=1112.376,305.088,-78.567,-177.827,10.511,149.530
C04935=1112.381,304.839,-78.535,-177.829,10.509,149.530
C04936=1112.385,304.593,-78.503,-177.832,10.507,149.531
C04937=1112.389,304.344,-78.470,-177.835,10.504,149.531
C04938=1112.393,304.096,-78.438,-177.839,10.501,149.531
C04939=1112.397,303.848,-78.406,-177.842,10.499,149.531
C04940=1112.401,303.600,-78.374,-177.845,10.496,149.531
C04941=1112.405,303.352,-78.343,-177.848,10.493,149.531
C04942=1112.409,303.104,-78.311,-177.851,10.491,149.532
C04943=1112.413,302.856,-78.278,-177.854,10.488,149.532
C04944=1112.418,302.609,-78.247,-177.857,10.486,149.532
C04945=1112.421,302.361,-78.215,-177.860,10.484,149.532
C04946=1112.426,302.112,-78.183,-177.863,10.481,149.532
C04947=1112.430,301.864,-78.151,-177.866,10.479,149.532
C04948=1112.434,301.617,-78.119,-177.869,10.476,149.533
C04949=1112.438,301.369,-78.087,-177.872,10.473,149.533
C04950=1112.442,301.121,-78.055,-177.876,10.471,149.533
C04951=1112.446,300.873,-78.023,-177.879,10.468,149.533
C04952=1112.450,300.625,-77.992,-177.882,10.466,149.533
C04953=1112.455,300.377,-77.959,-177.885,10.463,149.534
C04954=1112.459,300.129,-77.928,-177.888,10.461,149.534
C04955=1112.463,299.881,-77.896,-177.890,10.459,149.534
C04956=1112.466,299.633,-77.864,-177.894,10.456,149.534
C04957=1112.471,299.386,-77.832,-177.897,10.453,149.534
C04958=1112.475,299.138,-77.800,-177.900,10.451,149.535
C04959=1112.479,298.890,-77.768,-177.903,10.448,149.535
C04960=1112.483,298.642,-77.737,-177.906,10.446,149.535
C04961=1112.487,298.394,-77.706,-177.909,10.443,149.535
C04962=1112.491,298.146,-77.674,-177.913,10.441,149.535
C04963=1112.496,297.898,-77.642,-177.916,10.438,149.535
C04964=1112.499,297.650,-77.610,-177.918,10.436,149.536
C04965=1112.503,297.401,-77.579,-177.921,10.433,149.536
C04966=1112.508,297.154,-77.547,-177.925,10.431,149.536
C04967=1112.512,296.906,-77.515,-177.927,10.428,149.536
C04968=1112.516,296.659,-77.484,-177.931,10.426,149.536
C04969=1112.520,296.410,-77.453,-177.934,10.423,149.536
C04970=1112.524,296.162,-77.421,-177.937,10.421,149.537
C04971=1112.528,295.915,-77.389,-177.940,10.418,149.537
C04972=1112.532,295.666,-77.358,-177.943,10.415,149.537
C04973=1112.537,295.418,-77.326,-177.946,10.413,149.537
C04974=1112.541,295.170,-77.294,-177.949,10.411,149.537
C04975=1112.544,294.958,-77.268,-177.952,10.408,149.537
C04976=1112.548,294.745,-77.241,-177.954,10.406,149.538
C04977=1112.551,294.532,-77.214,-177.956,10.404,149.538
C04978=1112.554,294.320,-77.187,-177.960,10.402,149.538
C04979=1112.558,294.108,-77.160,-177.962,10.400,149.538
C04980=1112.562,293.895,-77.133,-177.964,10.398,149.538
C04981=1112.565,293.683,-77.106,-177.967,10.395,149.538
C04982=1112.569,293.470,-77.080,-177.970,10.393,149.539
C04983=1112.573,293.223,-77.048,-177.973,10.391,149.539
C04984=1112.577,292.974,-77.017,-177.976,10.388,149.539
C04985=1112.581,292.726,-76.985,-177.979,10.385,149.539
C04986=1112.585,292.478,-76.955,-177.983,10.383,149.539
C04987=1112.589,292.230,-76.923,-177.985,10.381,149.539
C04988=1112.593,291.982,-76.892,-177.988,10.378,149.539
C04989=1112.597,291.734,-76.860,-177.991,10.376,149.540
C04990=1112.602,291.486,-76.830,-177.994,10.373,149.540
C04991=1112.605,291.238,-76.798,-177.997,10.371,149.540
C04992=1112.609,290.990,-76.767,-178.000,10.368,149.540
C04993=1112.613,290.742,-76.736,-178.004,10.365,149.540
C04994=1112.618,290.494,-76.705,-178.007,10.363,149.541
C04995=1112.622,290.246,-76.674,-178.010,10.360,149.541
C04996=1112.626,289.998,-76.642,-178.012,10.358,149.541
C04997=1112.631,289.750,-76.612,-178.016,10.356,149.541
C04998=1112.634,289.502,-76.581,-178.019,10.353,149.541
C04999=1112.638,289.255,-76.549,-178.021,10.350,149.541
C05000=1112.642,289.006,-76.518,-178.025,10.348,149.542
C05001=1112.647,288.758,-76.488,-178.028,10.345,149.542
C05002=1112.651,288.509,-76.456,-178.031,10.343,149.542
C05003=1112.655,288.262,-76.425,-178.034,10.340,149.542
C05004=1112.658,288.014,-76.394,-178.037,10.338,149.542
C05005=1112.663,287.766,-76.364,-178.040,10.336,149.542
C05006=1112.668,287.518,-76.333,-178.043,10.333,149.543
C05007=1112.671,287.270,-76.301,-178.046,10.330,149.543
C05008=1112.675,287.022,-76.271,-178.049,10.328,149.543
C05009=1112.679,286.774,-76.240,-178.052,10.325,149.543
C05010=1112.684,286.526,-76.209,-178.055,10.322,149.543
C05011=1112.688,286.278,-76.178,-178.058,10.320,149.544
C05012=1112.692,286.029,-76.148,-178.061,10.317,149.544
C05013=1112.696,285.782,-76.116,-178.064,10.315,149.544
C05014=1112.700,285.533,-76.085,-178.067,10.313,149.544
C05015=1112.705,285.285,-76.054,-178.070,10.310,149.544
C05016=1112.709,285.038,-76.024,-178.073,10.308,149.544
C05017=1112.713,284.789,-75.993,-178.076,10.305,149.545
C05018=1112.717,284.541,-75.962,-178.080,10.302,149.545
C05019=1112.721,284.293,-75.932,-178.083,10.300,149.545
C05020=1112.725,284.045,-75.901,-178.085,10.297,149.545
C05021=1112.730,283.797,-75.870,-178.088,10.295,149.545
C05022=1112.734,283.549,-75.840,-178.091,10.293,149.545
C05023=1112.738,283.300,-75.809,-178.094,10.290,149.546
C05024=1112.741,283.053,-75.779,-178.097,10.287,149.546
C05025=1112.746,282.805,-75.748,-178.100,10.285,149.546
C05026=1112.751,282.557,-75.717,-178.104,10.282,149.546
C05027=1112.754,282.309,-75.687,-178.107,10.279,149.546
C05028=1112.759,282.061,-75.656,-178.110,10.277,149.547
C05029=1112.762,281.813,-75.626,-178.113,10.274,149.547
C05030=1112.767,281.564,-75.595,-178.116,10.273,149.547
C05031=1112.770,281.352,-75.569,-178.119,10.270,149.547
C05032=1112.774,281.139,-75.543,-178.121,10.268,149.547
C05033=1112.778,280.926,-75.517,-178.124,10.265,149.547
C05034=1112.781,280.714,-75.491,-178.127,10.263,149.548
C05035=1112.785,280.501,-75.465,-178.129,10.261,149.548
C05036=1112.789,280.288,-75.439,-178.132,10.259,149.548
C05037=1112.792,280.076,-75.412,-178.134,10.257,149.548
C05038=1112.796,279.863,-75.386,-178.137,10.254,149.548
C05039=1112.800,279.615,-75.356,-178.140,10.252,149.548
C05040=1112.804,279.367,-75.325,-178.143,10.249,149.548
C05041=1112.808,279.119,-75.295,-178.146,10.246,149.548
C05042=1112.812,278.871,-75.264,-178.150,10.244,149.549
C05043=1112.816,278.622,-75.235,-178.152,10.242,149.549
C05044=1112.820,278.375,-75.205,-178.155,10.239,149.549
C05045=1112.825,278.127,-75.174,-178.158,10.236,149.549
C05046=1112.829,277.878,-75.144,-178.161,10.234,149.549
C05047=1112.833,277.630,-75.113,-178.164,10.231,149.549
C05048=1112.837,277.382,-75.083,-178.167,10.228,149.549
C05049=1112.841,277.134,-75.054,-178.170,10.226,149.550
C05050=1112.846,276.886,-75.023,-178.173,10.223,149.550
C05051=1112.850,276.638,-74.993,-178.176,10.220,149.550
C05052=1112.854,276.389,-74.962,-178.179,10.217,149.550
C05053=1112.858,276.141,-74.932,-178.182,10.215,149.550
C05054=1112.862,275.893,-74.903,-178.185,10.212,149.550
C05055=1112.867,275.645,-74.872,-178.188,10.209,149.551
C05056=1112.871,275.397,-74.842,-178.191,10.207,149.551
C05057=1112.875,275.149,-74.812,-178.194,10.204,149.551
C05058=1112.879,274.900,-74.782,-178.196,10.202,149.551
C05059=1112.883,274.652,-74.752,-178.199,10.199,149.551
C05060=1112.887,274.404,-74.722,-178.202,10.196,149.551
C05061=1112.892,274.156,-74.691,-178.206,10.194,149.551
C05062=1112.896,273.908,-74.662,-178.209,10.191,149.551
C05063=1112.900,273.660,-74.632,-178.212,10.188,149.552
C05064=1112.904,273.412,-74.602,-178.215,10.186,149.552
C05065=1112.909,273.164,-74.572,-178.217,10.183,149.552
C05066=1112.913,272.916,-74.542,-178.220,10.181,149.552
C05067=1112.916,272.667,-74.512,-178.223,10.178,149.552
C05068=1112.920,272.419,-74.482,-178.226,10.175,149.552
C05069=1112.925,272.170,-74.452,-178.229,10.173,149.552
C05070=1112.929,271.923,-74.422,-178.232,10.170,149.552
C05071=1112.933,271.674,-74.392,-178.234,10.167,149.552
C05072=1112.937,271.426,-74.363,-178.237,10.164,149.552
C05073=1112.942,271.178,-74.332,-178.240,10.162,149.553
C05074=1112.946,270.930,-74.303,-178.243,10.160,149.553
C05075=1112.950,270.682,-74.273,-178.246,10.157,149.553
C05076=1112.955,270.433,-74.244,-178.249,10.155,149.553
C05077=1112.958,270.186,-74.214,-178.252,10.152,149.553
C05078=1112.963,269.938,-74.184,-178.254,10.150,149.553
C05079=1112.968,269.689,-74.154,-178.257,10.147,149.553
C05080=1112.972,269.441,-74.125,-178.260,10.144,149.553
C05081=1112.976,269.192,-74.095,-178.263,10.141,149.554
C05082=1112.980,268.945,-74.065,-178.266,10.139,149.554
C05083=1112.984,268.697,-74.036,-178.268,10.137,149.554
C05084=1112.988,268.448,-74.006,-178.271,10.134,149.554
C05085=1112.992,268.200,-73.977,-178.274,10.131,149.554
C05086=1112.996,267.952,-73.947,-178.277,10.128,149.554
C05087=1113.000,267.739,-73.921,-178.279,10.126,149.554
C05088=1113.004,267.526,-73.897,-178.282,10.124,149.554
C05089=1113.007,267.313,-73.871,-178.284,10.122,149.554
C05090=1113.011,267.100,-73.846,-178.286,10.120,149.554
C05091=1113.015,266.888,-73.820,-178.289,10.117,149.554
C05092=1113.018,266.674,-73.795,-178.291,10.115,149.555
C05093=1113.022,266.462,-73.769,-178.293,10.113,149.555
C05094=1113.026,266.249,-73.744,-178.296,10.111,149.555
C05095=1113.030,266.001,-73.715,-178.299,10.109,149.555
C05096=1113.034,265.752,-73.685,-178.301,10.107,149.555
C05097=1113.039,265.505,-73.656,-178.304,10.104,149.555
C05098=1113.043,265.257,-73.627,-178.307,10.101,149.555
C05099=1113.047,265.008,-73.597,-178.309,10.099,149.555
C05100=1113.051,264.760,-73.568,-178.312,10.096,149.556
C05101=1113.055,264.512,-73.538,-178.315,10.094,149.556
C05102=1113.060,264.264,-73.509,-178.318,10.091,149.556
C05103=1113.064,264.015,-73.479,-178.321,10.089,149.556
C05104=1113.068,263.767,-73.450,-178.324,10.086,149.556
C05105=1113.072,263.519,-73.421,-178.327,10.083,149.556
C05106=1113.076,263.270,-73.391,-178.331,10.081,149.557
C05107=1113.081,263.022,-73.362,-178.333,10.078,149.557
C05108=1113.085,262.774,-73.334,-178.336,10.075,149.557
C05109=1113.089,262.526,-73.304,-178.339,10.072,149.557
C05110=1113.093,262.278,-73.275,-178.342,10.070,149.557
C05111=1113.097,262.030,-73.245,-178.345,10.067,149.557
C05112=1113.102,261.781,-73.216,-178.349,10.064,149.557
C05113=1113.106,261.532,-73.187,-178.352,10.061,149.557
C05114=1113.110,261.284,-73.158,-178.355,10.058,149.558
C05115=1113.115,261.037,-73.129,-178.358,10.055,149.558
C05116=1113.119,260.788,-73.099,-178.361,10.053,149.558
C05117=1113.123,260.540,-73.071,-178.364,10.050,149.558
C05118=1113.127,260.291,-73.042,-178.367,10.047,149.558
C05119=1113.131,260.043,-73.012,-178.370,10.044,149.558
C05120=1113.136,259.796,-72.983,-178.372,10.041,149.558
C05121=1113.141,259.547,-72.954,-178.375,10.038,149.558
C05122=1113.144,259.299,-72.926,-178.378,10.036,149.558
C05123=1113.148,259.051,-72.896,-178.381,10.033,149.558
C05124=1113.153,258.802,-72.867,-178.383,10.031,149.558
C05125=1113.157,258.553,-72.838,-178.386,10.028,149.559
C05126=1113.161,258.305,-72.810,-178.389,10.025,149.559
C05127=1113.165,258.057,-72.781,-178.392,10.022,149.559
C05128=1113.170,257.809,-72.751,-178.395,10.020,149.559
C05129=1113.174,257.560,-72.722,-178.398,10.017,149.559
C05130=1113.178,257.313,-72.694,-178.401,10.014,149.559
C05131=1113.183,257.064,-72.665,-178.404,10.011,149.559
C05132=1113.187,256.816,-72.636,-178.406,10.008,149.559
C05133=1113.191,256.567,-72.608,-178.409,10.005,149.559
C05134=1113.195,256.319,-72.579,-178.412,10.003,149.559
C05135=1113.200,256.071,-72.550,-178.415,10.000,149.559
C05136=1113.203,255.823,-72.521,-178.416,9.998,149.559
C05137=1113.208,255.574,-72.492,-178.418,9.996,149.559
C05138=1113.213,255.326,-72.463,-178.420,9.994,149.559
C05139=1113.216,255.078,-72.435,-178.422,9.991,149.559
C05140=1113.220,254.829,-72.406,-178.424,9.989,149.559
C05141=1113.226,254.581,-72.377,-178.426,9.987,149.559
C05142=1113.229,254.333,-72.349,-178.428,9.985,149.559
C05143=1113.233,254.120,-72.324,-178.430,9.983,149.559
C05144=1113.236,253.907,-72.300,-178.432,9.982,149.559
C05145=1113.240,253.694,-72.275,-178.434,9.979,149.559
C05146=1113.245,253.481,-72.250,-178.436,9.977,149.559
C05147=1113.247,253.268,-72.225,-178.439,9.975,149.559
C05148=1113.252,253.056,-72.201,-178.441,9.973,149.560
C05149=1113.255,252.843,-72.177,-178.443,9.971,149.560
C05150=1113.259,252.629,-72.152,-178.445,9.969,149.560
C05151=1113.263,252.382,-72.123,-178.448,9.967,149.560
C05152=1113.267,252.133,-72.095,-178.451,9.965,149.560
C05153=1113.271,251.884,-72.067,-178.454,9.962,149.560
C05154=1113.276,251.637,-72.037,-178.457,9.959,149.561
C05155=1113.280,251.388,-72.009,-178.459,9.957,149.561
C05156=1113.284,251.139,-71.981,-178.463,9.955,149.561
C05157=1113.289,250.891,-71.953,-178.466,9.952,149.561
C05158=1113.293,250.643,-71.923,-178.470,9.949,149.561
C05159=1113.297,250.395,-71.895,-178.473,9.946,149.562
C05160=1113.302,250.146,-71.867,-178.476,9.944,149.562
C05161=1113.305,249.898,-71.839,-178.479,9.940,149.562
C05162=1113.310,249.649,-71.810,-178.483,9.938,149.562
C05163=1113.314,249.401,-71.782,-178.486,9.935,149.562
C05164=1113.318,249.153,-71.753,-178.490,9.931,149.563
C05165=1113.323,248.905,-71.725,-178.494,9.928,149.563
C05166=1113.327,248.656,-71.696,-178.498,9.925,149.563
C05167=1113.332,248.408,-71.668,-178.502,9.921,149.563
C05168=1113.336,248.159,-71.640,-178.505,9.918,149.563
C05169=1113.340,247.911,-71.612,-178.509,9.914,149.563
C05170=1113.344,247.663,-71.584,-178.513,9.911,149.564
C05171=1113.349,247.414,-71.555,-178.516,9.907,149.564
C05172=1113.353,247.166,-71.527,-178.518,9.905,149.564
C05173=1113.357,246.918,-71.499,-178.521,9.902,149.564
C05174=1113.362,246.669,-71.471,-178.523,9.900,149.563
C05175=1113.366,246.421,-71.443,-178.525,9.896,149.563
C05176=1113.370,246.173,-71.415,-178.527,9.894,149.563
C05177=1113.374,245.924,-71.386,-178.529,9.892,149.563
C05178=1113.379,245.676,-71.358,-178.531,9.889,149.563
C05179=1113.383,245.428,-71.330,-178.533,9.886,149.563
C05180=1113.388,245.179,-71.302,-178.536,9.884,149.563
C05181=1113.392,244.930,-71.274,-178.538,9.881,149.563
C05182=1113.396,244.682,-71.247,-178.541,9.878,149.563
C05183=1113.400,244.433,-71.218,-178.543,9.876,149.563
C05184=1113.405,244.186,-71.190,-178.545,9.873,149.563
C05185=1113.409,243.937,-71.162,-178.547,9.871,149.563
C05186=1113.413,243.689,-71.134,-178.550,9.868,149.563
C05187=1113.417,243.440,-71.105,-178.552,9.866,149.563
C05188=1113.422,243.192,-71.078,-178.554,9.863,149.563
C05189=1113.426,242.943,-71.050,-178.557,9.861,149.563
C05190=1113.430,242.695,-71.022,-178.559,9.858,149.563
C05191=1113.435,242.446,-70.994,-178.562,9.856,149.563
C05192=1113.439,242.198,-70.966,-178.564,9.853,149.563
C05193=1113.444,241.950,-70.939,-178.567,9.850,149.563
C05194=1113.447,241.701,-70.911,-178.570,9.848,149.563
C05195=1113.452,241.454,-70.883,-178.572,9.845,149.563
C05196=1113.456,241.205,-70.854,-178.575,9.843,149.563
C05197=1113.461,240.956,-70.827,-178.576,9.840,149.563
C05198=1113.465,240.708,-70.799,-178.579,9.838,149.564
C05199=1113.468,240.495,-70.775,-178.582,9.836,149.564
C05200=1113.472,240.282,-70.752,-178.584,9.833,149.564
C05201=1113.476,240.069,-70.728,-178.586,9.831,149.564
C05202=1113.480,239.856,-70.704,-178.588,9.829,149.564
C05203=1113.484,239.643,-70.680,-178.590,9.827,149.564
C05204=1113.488,239.430,-70.657,-178.592,9.825,149.564
C05205=1113.491,239.216,-70.633,-178.594,9.823,149.564
C05206=1113.494,239.004,-70.609,-178.597,9.821,149.564
C05207=1113.499,238.755,-70.581,-178.599,9.818,149.564
C05208=1113.503,238.507,-70.554,-178.602,9.815,149.564
C05209=1113.507,238.258,-70.526,-178.604,9.813,149.564
C05210=1113.511,238.010,-70.499,-178.607,9.810,149.564
C05211=1113.517,237.761,-70.471,-178.610,9.807,149.565
C05212=1113.521,237.513,-70.443,-178.612,9.805,149.564
C05213=1113.525,237.265,-70.415,-178.615,9.802,149.565
C05214=1113.529,237.016,-70.388,-178.618,9.799,149.565
C05215=1113.533,236.768,-70.360,-178.621,9.797,149.565
C05216=1113.538,236.519,-70.333,-178.623,9.795,149.565
C05217=1113.542,236.271,-70.305,-178.626,9.792,149.565
C05218=1113.546,236.022,-70.277,-178.629,9.789,149.565
C05219=1113.551,235.774,-70.250,-178.632,9.786,149.565
C05220=1113.555,235.526,-70.223,-178.634,9.784,149.565
C05221=1113.560,235.277,-70.195,-178.637,9.781,149.565
C05222=1113.564,235.029,-70.167,-178.640,9.778,149.565
C05223=1113.569,234.780,-70.140,-178.642,9.776,149.565
C05224=1113.573,234.531,-70.113,-178.645,9.773,149.566
C05225=1113.577,234.283,-70.085,-178.648,9.771,149.566
C05226=1113.582,234.035,-70.058,-178.651,9.768,149.566
C05227=1113.585,233.786,-70.030,-178.654,9.765,149.566
C05228=1113.590,233.538,-70.003,-178.656,9.762,149.566
C05229=1113.594,233.290,-69.976,-178.659,9.759,149.566
C05230=1113.599,233.041,-69.949,-178.662,9.757,149.566
C05231=1113.602,232.792,-69.921,-178.665,9.754,149.566
C05232=1113.607,232.544,-69.894,-178.668,9.751,149.566
C05233=1113.612,232.295,-69.867,-178.670,9.748,149.566
C05234=1113.616,232.048,-69.839,-178.673,9.745,149.566
C05235=1113.620,231.798,-69.812,-178.676,9.743,149.567
C05236=1113.625,231.550,-69.785,-178.679,9.740,149.567
C05237=1113.629,231.302,-69.758,-178.682,9.737,149.567
C05238=1113.633,231.053,-69.731,-178.685,9.734,149.567
C05239=1113.638,230.805,-69.704,-178.688,9.731,149.567
C05240=1113.642,230.556,-69.676,-178.690,9.728,149.567
C05241=1113.646,230.308,-69.649,-178.693,9.725,149.567
C05242=1113.651,230.059,-69.622,-178.696,9.723,149.567
C05243=1113.655,229.811,-69.596,-178.699,9.719,149.567
C05244=1113.660,229.562,-69.568,-178.702,9.716,149.567
C05245=1113.664,229.313,-69.541,-178.705,9.713,149.567
C05246=1113.668,229.065,-69.514,-178.708,9.710,149.567
C05247=1113.673,228.816,-69.487,-178.711,9.707,149.567
C05248=1113.677,228.569,-69.460,-178.713,9.704,149.567
C05249=1113.681,228.320,-69.433,-178.716,9.702,149.567
C05250=1113.686,228.072,-69.406,-178.719,9.698,149.567
C05251=1113.689,227.823,-69.379,-178.722,9.695,149.567
C05252=1113.694,227.574,-69.352,-178.725,9.692,149.567
C05253=1113.698,227.326,-69.325,-178.728,9.689,149.567
C05254=1113.703,227.077,-69.298,-178.730,9.686,149.567
C05255=1113.706,226.864,-69.275,-178.733,9.683,149.567
C05256=1113.710,226.651,-69.252,-178.735,9.681,149.567
C05257=1113.714,226.437,-69.229,-178.738,9.678,149.567
C05258=1113.718,226.224,-69.206,-178.739,9.675,149.567
C05259=1113.722,226.012,-69.184,-178.742,9.672,149.567
C05260=1113.726,225.799,-69.160,-178.744,9.670,149.567
C05261=1113.729,225.586,-69.137,-178.747,9.667,149.567
C05262=1113.733,225.372,-69.114,-178.749,9.665,149.567
C05263=1113.737,225.124,-69.087,-178.751,9.662,149.567
C05264=1113.742,224.875,-69.060,-178.754,9.659,149.567
C05265=1113.747,224.627,-69.033,-178.756,9.656,149.567
C05266=1113.751,224.378,-69.008,-178.759,9.652,149.567
C05267=1113.755,224.129,-68.980,-178.761,9.649,149.567
C05268=1113.759,223.881,-68.954,-178.764,9.646,149.567
C05269=1113.763,223.632,-68.927,-178.766,9.643,149.567
C05270=1113.767,223.384,-68.900,-178.769,9.640,149.567
C05271=1113.772,223.135,-68.874,-178.772,9.637,149.567
C05272=1113.777,222.886,-68.847,-178.774,9.634,149.567
C05273=1113.781,222.638,-68.820,-178.777,9.631,149.567
C05274=1113.786,222.390,-68.793,-178.779,9.628,149.566
C05275=1113.790,222.141,-68.768,-178.782,9.624,149.566
C05276=1113.794,221.892,-68.740,-178.784,9.621,149.566
C05277=1113.798,221.644,-68.714,-178.787,9.618,149.566
C05278=1113.803,221.395,-68.688,-178.789,9.615,149.566
C05279=1113.807,221.147,-68.661,-178.792,9.612,149.566
C05280=1113.812,220.898,-68.634,-178.794,9.609,149.566
C05281=1113.816,220.650,-68.608,-178.797,9.606,149.566
C05282=1113.821,220.401,-68.581,-178.799,9.603,149.566
C05283=1113.825,220.152,-68.556,-178.802,9.600,149.566
C05284=1113.830,219.904,-68.528,-178.804,9.596,149.566
C05285=1113.834,219.656,-68.502,-178.806,9.594,149.566
C05286=1113.838,219.407,-68.476,-178.808,9.591,149.565
C05287=1113.842,219.158,-68.449,-178.811,9.588,149.565
C05288=1113.847,218.910,-68.423,-178.813,9.584,149.565
C05289=1113.851,218.661,-68.396,-178.815,9.581,149.565
C05290=1113.856,218.413,-68.371,-178.818,9.578,149.565
C05291=1113.860,218.165,-68.345,-178.820,9.576,149.565
C05292=1113.865,217.916,-68.318,-178.822,9.572,149.565
C05293=1113.869,217.667,-68.292,-178.825,9.569,149.565
C05294=1113.874,217.418,-68.265,-178.827,9.566,149.565
C05295=1113.878,217.170,-68.239,-178.830,9.563,149.565
C05296=1113.882,216.921,-68.213,-178.831,9.560,149.564
C05297=1113.887,216.672,-68.187,-178.834,9.557,149.564
C05298=1113.891,216.424,-68.160,-178.836,9.554,149.564
C05299=1113.895,216.175,-68.135,-178.838,9.551,149.564
C05300=1113.899,215.927,-68.108,-178.841,9.548,149.564
C05301=1113.904,215.678,-68.082,-178.843,9.545,149.564
C05302=1113.909,215.430,-68.056,-178.845,9.543,149.564
C05303=1113.913,215.182,-68.030,-178.847,9.539,149.564
C05304=1113.918,214.933,-68.004,-178.850,9.536,149.564
C05305=1113.922,214.684,-67.978,-178.851,9.534,149.563
C05306=1113.926,214.436,-67.951,-178.854,9.531,149.563
C05307=1113.930,214.187,-67.926,-178.856,9.527,149.563
C05308=1113.935,213.938,-67.899,-178.858,9.525,149.563
C05309=1113.939,213.689,-67.873,-178.860,9.522,149.563
C05310=1113.944,213.441,-67.847,-178.862,9.519,149.563
C05311=1113.948,213.228,-67.825,-178.864,9.516,149.563
C05312=1113.951,213.014,-67.802,-178.866,9.514,149.563
C05313=1113.955,212.802,-67.781,-178.869,9.511,149.563
C05314=1113.959,212.588,-67.758,-178.871,9.509,149.563
C05315=1113.962,212.375,-67.736,-178.874,9.506,149.563
C05316=1113.966,212.161,-67.713,-178.876,9.503,149.563
C05317=1113.970,211.948,-67.691,-178.879,9.501,149.563
C05318=1113.974,211.735,-67.669,-178.881,9.497,149.563
C05319=1113.979,211.486,-67.642,-178.884,9.494,149.563
C05320=1113.983,211.238,-67.617,-178.887,9.492,149.563
C05321=1113.988,210.989,-67.591,-178.889,9.489,149.563
C05322=1113.992,210.740,-67.566,-178.892,9.485,149.563
C05323=1113.996,210.492,-67.540,-178.895,9.483,149.563
C05324=1114.000,210.243,-67.514,-178.897,9.480,149.563
C05325=1114.005,209.995,-67.489,-178.900,9.477,149.563
C05326=1114.010,209.746,-67.462,-178.903,9.474,149.563
C05327=1114.014,209.497,-67.436,-178.906,9.471,149.563
C05328=1114.018,209.248,-67.410,-178.908,9.468,149.563
C05329=1114.023,209.000,-67.385,-178.911,9.465,149.563
C05330=1114.027,208.752,-67.359,-178.914,9.462,149.563
C05331=1114.032,208.503,-67.333,-178.916,9.459,149.563
C05332=1114.036,208.254,-67.308,-178.920,9.456,149.563
C05333=1114.041,208.006,-67.282,-178.923,9.453,149.563
C05334=1114.045,207.757,-67.256,-178.926,9.450,149.563
C05335=1114.049,207.508,-67.231,-178.928,9.447,149.564
C05336=1114.054,207.260,-67.206,-178.931,9.444,149.564
C05337=1114.058,207.011,-67.180,-178.934,9.442,149.564
C05338=1114.063,206.762,-67.154,-178.937,9.439,149.564
C05339=1114.067,206.514,-67.129,-178.940,9.436,149.564
C05340=1114.072,206.265,-67.103,-178.943,9.433,149.564
C05341=1114.076,206.016,-67.078,-178.945,9.430,149.564
C05342=1114.081,205.768,-67.052,-178.948,9.427,149.564
C05343=1114.085,205.519,-67.026,-178.951,9.424,149.564
C05344=1114.089,205.270,-67.001,-178.954,9.422,149.564
C05345=1114.094,205.022,-66.976,-178.957,9.419,149.564
C05346=1114.099,204.773,-66.950,-178.960,9.416,149.565
C05347=1114.103,204.524,-66.925,-178.963,9.413,149.565
C05348=1114.108,204.276,-66.899,-178.966,9.410,149.565
C05349=1114.112,204.027,-66.874,-178.968,9.407,149.565
C05350=1114.116,203.778,-66.848,-178.971,9.404,149.565
C05351=1114.121,203.530,-66.823,-178.975,9.401,149.565
C05352=1114.125,203.281,-66.797,-178.978,9.398,149.565
C05353=1114.130,203.033,-66.773,-178.980,9.395,149.565
C05354=1114.134,202.784,-66.747,-178.983,9.392,149.565
C05355=1114.138,202.535,-66.722,-178.986,9.390,149.565
C05356=1114.143,202.286,-66.697,-178.989,9.387,149.565
C05357=1114.148,202.037,-66.671,-178.991,9.384,149.566
C05358=1114.152,201.789,-66.646,-178.994,9.381,149.566
C05359=1114.156,201.540,-66.621,-178.997,9.378,149.566
C05360=1114.160,201.291,-66.596,-179.000,9.375,149.566
C05361=1114.166,201.043,-66.571,-179.003,9.372,149.566
C05362=1114.170,200.794,-66.545,-179.006,9.369,149.566
C05363=1114.175,200.545,-66.521,-179.009,9.366,149.566
C05364=1114.178,200.297,-66.495,-179.012,9.363,149.566
C05365=1114.183,200.049,-66.470,-179.014,9.360,149.566
C05366=1114.188,199.799,-66.445,-179.017,9.357,149.566
C05367=1114.192,199.586,-66.424,-179.020,9.354,149.566
C05368=1114.195,199.373,-66.402,-179.023,9.351,149.566
C05369=1114.199,199.159,-66.381,-179.025,9.349,149.566
C05370=1114.203,198.945,-66.359,-179.027,9.346,149.566
C05371=1114.207,198.733,-66.337,-179.030,9.344,149.566
C05372=1114.211,198.519,-66.316,-179.032,9.341,149.566
C05373=1114.215,198.305,-66.295,-179.035,9.338,149.566
C05374=1114.219,198.092,-66.274,-179.037,9.336,149.566
C05375=1114.223,197.844,-66.248,-179.040,9.332,149.566
C05376=1114.228,197.595,-66.224,-179.043,9.329,149.567
C05377=1114.232,197.346,-66.198,-179.046,9.326,149.566
C05378=1114.236,197.098,-66.174,-179.048,9.323,149.566
C05379=1114.241,196.848,-66.149,-179.052,9.319,149.567
C05380=1114.246,196.600,-66.123,-179.054,9.316,149.567
C05381=1114.249,196.351,-66.099,-179.057,9.313,149.566
C05382=1114.255,196.102,-66.074,-179.059,9.310,149.566
C05383=1114.258,195.854,-66.049,-179.061,9.307,149.566
C05384=1114.263,195.605,-66.025,-179.063,9.305,149.566
C05385=1114.268,195.356,-65.999,-179.065,9.302,149.566
C05386=1114.272,195.107,-65.975,-179.067,9.299,149.566
C05387=1114.277,194.859,-65.950,-179.069,9.296,149.566
C05388=1114.281,194.610,-65.926,-179.071,9.293,149.566
C05389=1114.286,194.361,-65.901,-179.073,9.291,149.565
C05390=1114.290,194.112,-65.876,-179.075,9.288,149.565
C05391=1114.294,193.864,-65.851,-179.077,9.286,149.565
C05392=1114.300,193.615,-65.826,-179.079,9.282,149.565
C05393=1114.303,193.366,-65.802,-179.081,9.280,149.565
C05394=1114.309,193.118,-65.777,-179.083,9.277,149.565
C05395=1114.312,192.869,-65.753,-179.085,9.274,149.565
C05396=1114.317,192.620,-65.728,-179.088,9.271,149.565
C05397=1114.322,192.372,-65.703,-179.089,9.269,149.565
C05398=1114.326,192.123,-65.678,-179.092,9.266,149.565
C05399=1114.330,191.874,-65.654,-179.094,9.263,149.565
C05400=1114.336,191.625,-65.630,-179.096,9.260,149.565
C05401=1114.339,191.376,-65.605,-179.098,9.258,149.565
C05402=1114.345,191.128,-65.581,-179.101,9.255,149.565
C05403=1114.348,190.879,-65.556,-179.103,9.252,149.564
C05404=1114.353,190.630,-65.531,-179.105,9.249,149.564
C05405=1114.358,190.381,-65.507,-179.107,9.247,149.564
C05406=1114.362,190.132,-65.482,-179.110,9.244,149.564
C05407=1114.367,189.884,-65.458,-179.111,9.241,149.564
C05408=1114.371,189.635,-65.434,-179.114,9.238,149.564
C05409=1114.376,189.386,-65.409,-179.116,9.236,149.564
C05410=1114.380,189.137,-65.385,-179.118,9.233,149.564
C05411=1114.385,188.889,-65.360,-179.121,9.230,149.564
C05412=1114.390,188.640,-65.336,-179.123,9.227,149.564
C05413=1114.393,188.391,-65.312,-179.125,9.224,149.564
C05414=1114.399,188.142,-65.287,-179.127,9.222,149.564
C05415=1114.403,187.894,-65.263,-179.130,9.219,149.564
C05416=1114.407,187.644,-65.238,-179.132,9.216,149.564
C05417=1114.412,187.396,-65.214,-179.134,9.213,149.564
C05418=1114.416,187.148,-65.190,-179.137,9.210,149.564
C05419=1114.421,186.899,-65.165,-179.139,9.207,149.564
C05420=1114.425,186.650,-65.141,-179.141,9.205,149.564
C05421=1114.430,186.401,-65.117,-179.144,9.202,149.564
C05422=1114.435,186.152,-65.093,-179.146,9.199,149.564
C05423=1114.438,185.939,-65.072,-179.148,9.196,149.564
C05424=1114.442,185.725,-65.051,-179.150,9.194,149.564
C05425=1114.446,185.512,-65.030,-179.152,9.192,149.564
C05426=1114.450,185.298,-65.010,-179.154,9.189,149.563
C05427=1114.454,185.085,-64.989,-179.156,9.186,149.563
C05428=1114.457,184.871,-64.968,-179.158,9.184,149.563
C05429=1114.462,184.658,-64.947,-179.160,9.182,149.563
C05430=1114.466,184.444,-64.926,-179.162,9.179,149.563
C05431=1114.470,184.196,-64.902,-179.164,9.176,149.563
C05432=1114.474,183.946,-64.879,-179.167,9.173,149.563
C05433=1114.479,183.698,-64.855,-179.170,9.170,149.563
C05434=1114.484,183.449,-64.830,-179.172,9.167,149.563
C05435=1114.488,183.201,-64.806,-179.175,9.164,149.563
C05436=1114.493,182.952,-64.782,-179.177,9.162,149.563
C05437=1114.497,182.703,-64.758,-179.179,9.159,149.563
C05438=1114.501,182.454,-64.734,-179.182,9.156,149.563
C05439=1114.507,182.205,-64.710,-179.184,9.152,149.563
C05440=1114.511,181.956,-64.686,-179.187,9.149,149.563
C05441=1114.515,181.708,-64.662,-179.189,9.146,149.563
C05442=1114.520,181.459,-64.638,-179.192,9.143,149.563
C05443=1114.524,181.210,-64.614,-179.194,9.140,149.563
C05444=1114.529,180.961,-64.591,-179.197,9.137,149.563
C05445=1114.534,180.712,-64.566,-179.200,9.134,149.563
C05446=1114.538,180.464,-64.542,-179.202,9.131,149.563
C05447=1114.543,180.215,-64.519,-179.205,9.128,149.563
C05448=1114.547,179.966,-64.494,-179.207,9.124,149.563
C05449=1114.552,179.717,-64.471,-179.210,9.121,149.563
C05450=1114.556,179.469,-64.447,-179.212,9.118,149.563
C05451=1114.560,179.219,-64.423,-179.215,9.115,149.563
